KUKA KRL program: MyProgram_116().src

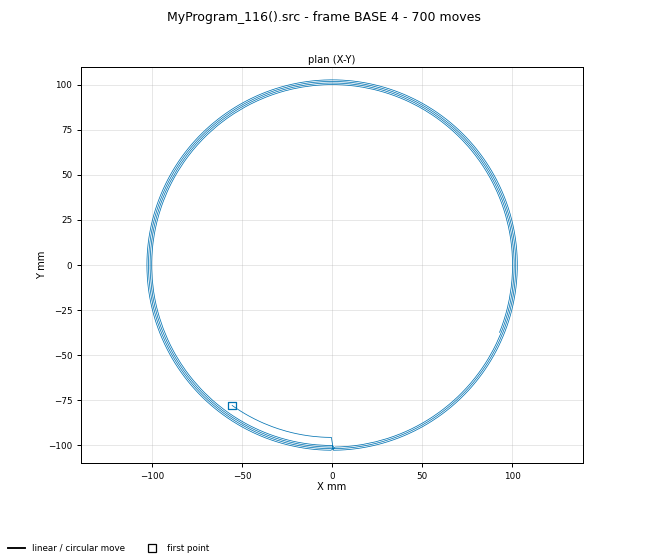
[picture p0: tool path of MyProgram_116().src in frame BASE 4, 700 of 700 moves have a stored position in this frame; points joined in program order, loops and branches not executed]
&ACCESS RVP
&REL 1
&PARAM TEMPLATE = C:\KRC\Roboter\Template\vorgabe
&PARAM EDITMASK = *
DEF MyProgram_116()
; ---- Setting reference (Base) ----
$BASE = BASE_DATA[4]

; --------------------------
; ---- Setting tool (TCP) ----
$TOOL = TOOL_DATA[3]
; --------------------------

$VEL.CP = VEL_APROX_PRINT
Startdeposition()
$VEL.CP = VEL_PRINT
LIN {X -55.4095,Y -77.8597,Z 99,A -129.4251,B 24.9347,C -1.8661,E1 24.9084,E2 214.7041} C_DIS
LIN {X -53.0962,Y -79.4573,Z 99,A -127.8078,B 24.9351,C -1.8611,E1 24.9121,E2 213.0935} C_DIS
LIN {X -50.3768,Y -81.2071,Z 99,A -125.8595,B 24.9353,C -1.8584,E1 24.9167,E2 211.1452} C_DIS
LIN {X -48.3524,Y -82.4286,Z 99,A -124.4407,B 24.9353,C -1.8564,E1 24.9201,E2 209.7269} C_DIS
LIN {X -46.0787,Y -83.7223,Z 99,A -122.868,B 24.9355,C -1.8544,E1 24.9239,E2 208.1545} C_DIS
LIN {X -42.9713,Y -85.3589,Z 99,A -120.7555,B 24.9357,C -1.8519,E1 24.9292,E2 206.042} C_DIS
LIN {X -40.0549,Y -86.7642,Z 99,A -118.7797,B 24.9357,C -1.8509,E1 24.9341,E2 204.0638} C_DIS
LIN {X -37.783,Y -87.778,Z 99,A -117.3046,B 24.9359,C -1.8487,E1 24.9379,E2 202.5903} C_DIS
LIN {X -35.4871,Y -88.7318,Z 99,A -115.8209,B 24.9361,C -1.847,E1 24.9417,E2 201.1074} C_DIS
LIN {X -33.3081,Y -89.5725,Z 99,A -114.4196,B 24.9361,C -1.8457,E1 24.9454,E2 199.7061} C_DIS
LIN {X -29.9786,Y -90.7411,Z 99,A -112.2978,B 24.9363,C -1.8442,E1 24.951,E2 197.5839} C_DIS
LIN {X -27.7453,Y -91.4487,Z 99,A -110.8917,B 24.9363,C -1.8432,E1 24.9548,E2 196.1778} C_DIS
LIN {X -25.4955,Y -92.1013,Z 99,A -109.4857,B 24.9363,C -1.8423,E1 24.9585,E2 194.7716} C_DIS
LIN {X -22.0782,Y -92.9797,Z 99,A -107.3681,B 24.9365,C -1.8412,E1 24.9643,E2 192.6536} C_DIS
LIN {X -19.7944,Y -93.4925,Z 99,A -105.9617,B 24.9365,C -1.8407,E1 24.9681,E2 191.2467} C_DIS
LIN {X -16.3468,Y -94.1565,Z 99,A -103.8547,B 24.9365,C -1.84,E1 24.9739,E2 189.1391} C_DIS
LIN {X -13.1497,Y -94.6546,Z 99,A -101.8803,B 24.9365,C -1.8407,E1 24.9794,E2 187.1612} C_DIS
LIN {X -10.5338,Y -94.9827,Z 99,A -100.3324,B 24.9365,C -1.8393,E1 24.9837,E2 185.6157} C_DIS
LIN {X -8.2054,Y -95.2121,Z 99,A -98.9301,B 24.9365,C -1.8393,E1 24.9876,E2 184.2129} C_DIS
LIN {X -6.146,Y -95.3659,Z 99,A -97.6617,B 24.9365,C -1.8403,E1 24.9911,E2 182.9415} C_DIS
LIN {X -3.7954,Y -95.4883,Z 99,A -96.2517,B 24.9365,C -1.8404,E1 24.995,E2 181.5309} C_DIS
LIN {X -0.3905,Y -95.5626,Z 99,A -94.2196,B 24.9365,C -1.8404,E1 25.0007,E2 179.4987} C_DIS
LIN {X -0.3905,Y -95.5626,Z 99,A -94.2196,B 24.9365,C -1.8404,E1 25.0007,E2 179.4987} C_DIS
Enddeposition()
LIN {X 0.7142,Y -102.6796,Z 100,A -93.2749,B 24.9435,C -1.7358,E1 25.0027,E2 178.8022} C_DIS
Startdeposition()
$VEL.CP = VEL_PRINT
LIN {X 4.3511,Y -102.5901,Z 100,A -91.2947,B 24.9436,C -1.7345,E1 25.0082,E2 176.8254} C_DIS
LIN {X 7.5539,Y -102.406,Z 100,A -89.3348,B 24.9431,C -1.7419,E1 25.0137,E2 174.8488} C_DIS
LIN {X 10.7491,Y -102.1182,Z 100,A -87.6564,B 24.9434,C -1.7386,E1 25.0183,E2 173.1795} C_DIS
LIN {X 13.8193,Y -101.7501,Z 100,A -86.0246,B 24.9435,C -1.7359,E1 25.0228,E2 171.5552} C_DIS
LIN {X 16.3122,Y -101.3803,Z 100,A -84.614,B 24.9435,C -1.7371,E1 25.0267,E2 170.1431} C_DIS
LIN {X 19.3571,Y -100.8413,Z 100,A -82.8685,B 24.9433,C -1.7394,E1 25.0315,E2 168.3943} C_DIS
LIN {X 22.4982,Y -100.1892,Z 100,A -80.9107,B 24.9428,C -1.7476,E1 25.0369,E2 166.4195} C_DIS
LIN {X 25.5043,Y -99.4645,Z 100,A -79.3897,B 24.9432,C -1.7413,E1 25.041,E2 164.9158} C_DIS
LIN {X 28.0492,Y -98.777,Z 100,A -77.8313,B 24.9428,C -1.7463,E1 25.0452,E2 163.348} C_DIS
LIN {X 31.0113,Y -97.8895,Z 100,A -76.2013,B 24.943,C -1.7445,E1 25.0495,E2 161.7252} C_DIS
LIN {X 33.944,Y -96.9096,Z 100,A -74.4511,B 24.9428,C -1.7477,E1 25.0542,E2 159.9708} C_DIS
LIN {X 36.9556,Y -95.8037,Z 100,A -72.5014,B 24.9422,C -1.7565,E1 25.0593,E2 158.0045} C_DIS
LIN {X 39.8227,Y -94.6457,Z 100,A -70.9753,B 24.9425,C -1.751,E1 25.0632,E2 156.495} C_DIS
LIN {X 42.2392,Y -93.5923,Z 100,A -69.4185,B 24.9422,C -1.7567,E1 25.0672,E2 154.9285} C_DIS
LIN {X 45.5515,Y -92.0256,Z 100,A -67.3851,B 24.942,C -1.7596,E1 25.0723,E2 152.8938} C_DIS
LIN {X 48.405,Y -90.5594,Z 100,A -65.6879,B 24.942,C -1.7588,E1 25.0765,E2 151.2031} C_DIS
LIN {X 50.6129,Y -89.3442,Z 100,A -64.2871,B 24.9419,C -1.7611,E1 25.0799,E2 149.801} C_DIS
LIN {X 53.2791,Y -87.7781,Z 100,A -62.5689,B 24.9417,C -1.764,E1 25.084,E2 148.0812} C_DIS
LIN {X 55.5149,Y -86.3815,Z 100,A -61.0131,B 24.9413,C -1.7703,E1 25.0877,E2 146.5155} C_DIS
LIN {X 58.5615,Y -84.3458,Z 100,A -59.0387,B 24.9412,C -1.7715,E1 25.0923,E2 144.5449} C_DIS
LIN {X 61.1689,Y -82.4768,Z 100,A -57.286,B 24.941,C -1.7737,E1 25.0962,E2 142.7933} C_DIS
LIN {X 63.5218,Y -80.6764,Z 100,A -55.5728,B 24.9406,C -1.7798,E1 25.1,E2 141.072} C_DIS
LIN {X 66.1114,Y -78.5706,Z 100,A -53.587,B 24.94,C -1.789,E1 25.1043,E2 139.0721} C_DIS
LIN {X 68.5323,Y -76.4656,Z 100,A -51.9152,B 24.94,C -1.7883,E1 25.1078,E2 137.4086} C_DIS
LIN {X 71.0991,Y -74.0852,Z 100,A -49.9841,B 24.9398,C -1.792,E1 25.1117,E2 135.4766} C_DIS
LIN {X 73.4943,Y -71.7122,Z 100,A -48.191,B 24.9398,C -1.7929,E1 25.1153,E2 133.6889} C_DIS
LIN {X 75.6188,Y -69.4655,Z 100,A -46.4342,B 24.9394,C -1.7986,E1 25.1186,E2 131.9264} C_DIS
LIN {X 77.7534,Y -67.0706,Z 100,A -44.4949,B 24.9386,C -1.8094,E1 25.1222,E2 129.9704} C_DIS
LIN {X 79.7362,Y -64.6978,Z 100,A -42.9791,B 24.9389,C -1.8053,E1 25.1249,E2 128.4713} C_DIS
LIN {X 81.2999,Y -62.7215,Z 100,A -41.5516,B 24.9386,C -1.8099,E1 25.1273,E2 127.0396} C_DIS
LIN {X 83.2212,Y -60.1522,Z 100,A -39.6726,B 24.938,C -1.8185,E1 25.1304,E2 125.1494} C_DIS
LIN {X 84.9931,Y -57.6181,Z 100,A -38.0863,B 24.938,C -1.8175,E1 25.1329,E2 123.5732} C_DIS
LIN {X 86.3815,Y -55.5149,Z 100,A -36.6593,B 24.9377,C -1.8224,E1 25.1351,E2 122.1418} C_DIS
LIN {X 88.0752,Y -52.7903,Z 100,A -34.7097,B 24.9369,C -1.8341,E1 25.138,E2 120.1745} C_DIS
LIN {X 89.6231,Y -50.1134,Z 100,A -33.1655,B 24.9371,C -1.8316,E1 25.1401,E2 118.6442} C_DIS
LIN {X 91.1466,Y -47.2901,Z 100,A -31.4161,B 24.9369,C -1.8352,E1 25.1424,E2 116.8955} C_DIS
LIN {X 92.5275,Y -44.5234,Z 100,A -29.702,B 24.9365,C -1.8399,E1 25.1445,E2 115.1795} C_DIS
LIN {X 93.5923,Y -42.2392,Z 100,A -28.2755,B 24.9362,C -1.845,E1 25.1462,E2 113.7487} C_DIS
LIN {X 94.8679,Y -39.2956,Z 100,A -26.5265,B 24.9359,C -1.8488,E1 25.1481,E2 112.0004} C_DIS
LIN {X 95.8037,Y -36.9556,Z 100,A -24.93,B 24.9351,C -1.8611,E1 25.1497,E2 110.3838} C_DIS
LIN {X 96.9096,Y -33.944,Z 100,A -23.2609,B 24.9351,C -1.8616,E1 25.1513,E2 108.7228} C_DIS
LIN {X 97.8895,Y -31.0113,Z 100,A -21.4381,B 24.9344,C -1.8711,E1 25.1528,E2 106.888} C_DIS
LIN {X 98.777,Y -28.0492,Z 100,A -19.8946,B 24.9345,C -1.8689,E1 25.154,E2 105.3584} C_DIS
LIN {X 99.6069,Y -24.9502,Z 100,A -17.9906,B 24.9338,C -1.8794,E1 25.1554,E2 103.4408} C_DIS
LIN {X 100.3112,Y -21.9393,Z 100,A -16.4325,B 24.9338,C -1.8779,E1 25.1563,E2 101.8951} C_DIS
LIN {X 100.8413,Y -19.3571,Z 100,A -14.8812,B 24.9333,C -1.886,E1 25.1572,E2 100.3339} C_DIS
LIN {X 101.4677,Y -15.7469,Z 100,A -12.8865,B 24.933,C -1.8905,E1 25.1581,E2 98.3403} C_DIS
LIN {X 101.912,Y -12.5696,Z 100,A -10.9641,B 24.9322,C -1.9018,E1 25.1588,E2 96.4025} C_DIS
LIN {X 102.253,Y -9.3797,Z 100,A -9.2954,B 24.9322,C -1.9025,E1 25.1592,E2 94.7421} C_DIS
LIN {X 102.5226,Y -5.7255,Z 100,A -7.3261,B 24.9319,C -1.9059,E1 25.1596,E2 92.7763} C_DIS
LIN {X 102.6533,Y -2.52,Z 100,A -5.5778,B 24.9316,C -1.9099,E1 25.1598,E2 91.029} C_DIS
LIN {X 102.6658,Y 1.8399,Z 100,A -3.1348,B 24.931,C -1.9183,E1 25.1598,E2 88.5808} C_DIS
LIN {X 102.5606,Y 5.0385,Z 100,A -1.2021,B 24.9302,C -1.9301,E1 25.1595,E2 86.6317} C_DIS
LIN {X 102.3604,Y 8.1242,Z 100,A 0.3545,B 24.9302,C -1.9286,E1 25.1592,E2 85.0879} C_DIS
LIN {X 102.0586,Y 11.3181,Z 100,A 2.103,B 24.93,C -1.9325,E1 25.1587,E2 83.3405} C_DIS
LIN {X 101.6696,Y 14.3857,Z 100,A 3.8167,B 24.9296,C -1.9375,E1 25.1581,E2 81.6251} C_DIS
LIN {X 101.286,Y 16.8765,Z 100,A 5.2133,B 24.9293,C -1.9416,E1 25.1574,E2 80.2272} C_DIS
LIN {X 100.8413,Y 19.3571,Z 100,A 6.6896,B 24.9288,C -1.9489,E1 25.1567,E2 78.7422} C_DIS
LIN {X 100.1892,Y 22.4982,Z 100,A 8.5878,B 24.9281,C -1.959,E1 25.1556,E2 76.8314} C_DIS
LIN {X 99.4645,Y 25.5043,Z 100,A 10.1428,B 24.9281,C -1.9572,E1 25.1545,E2 75.2894} C_DIS
LIN {X 98.6211,Y 28.5996,Z 100,A 12.0792,B 24.9273,C -1.9687,E1 25.153,E2 73.337} C_DIS
LIN {X 97.6777,Y 31.6659,Z 100,A 13.7497,B 24.9273,C -1.9691,E1 25.1516,E2 71.6749} C_DIS
LIN {X 96.4857,Y 35.1307,Z 100,A 15.7578,B 24.927,C -1.9737,E1 25.1498,E2 69.6673} C_DIS
LIN {X 95.343,Y 38.1284,Z 100,A 17.6692,B 24.9262,C -1.9839,E1 25.1478,E2 67.7424} C_DIS
LIN {X 94.1036,Y 41.0875,Z 100,A 19.339,B 24.9262,C -1.9842,E1 25.146,E2 66.0812} C_DIS
LIN {X 92.8255,Y 43.9032,Z 100,A 21.1632,B 24.9255,C -1.9931,E1 25.1438,E2 64.2458} C_DIS
LIN {X 91.3057,Y 46.9788,Z 100,A 22.9045,B 24.9257,C -1.9913,E1 25.1416,E2 62.518} C_DIS
LIN {X 89.9586,Y 49.5127,Z 100,A 24.6576,B 24.9249,C -2.0019,E1 25.1393,E2 60.749} C_DIS
LIN {X 88.4253,Y 52.1979,Z 100,A 26.173,B 24.9252,C -1.9979,E1 25.1372,E2 59.2508} C_DIS
LIN {X 87.1177,Y 54.3523,Z 100,A 27.6426,B 24.9247,C -2.0043,E1 25.135,E2 57.7738} C_DIS
LIN {X 85.3788,Y 57.0483,Z 100,A 29.3516,B 24.9246,C -2.0055,E1 25.1324,E2 56.0704} C_DIS
LIN {X 83.9531,Y 59.1264,Z 100,A 30.9333,B 24.9238,C -2.0163,E1 25.1298,E2 54.4711} C_DIS
LIN {X 82.1332,Y 61.6263,Z 100,A 32.4958,B 24.924,C -2.0139,E1 25.1273,E2 52.9216} C_DIS
LIN {X 80.1694,Y 64.1632,Z 100,A 34.2472,B 24.9237,C -2.0166,E1 25.1242,E2 51.1721} C_DIS
LIN {X 78.5706,Y 66.1114,Z 100,A 35.7514,B 24.9232,C -2.0239,E1 25.1215,E2 49.6576} C_DIS
LIN {X 76.5429,Y 68.4459,Z 100,A 37.3928,B 24.9232,C -2.0244,E1 25.1185,E2 48.0222} C_DIS
LIN {X 74.3688,Y 70.805,Z 100,A 39.145,B 24.923,C -2.0268,E1 25.1152,E2 46.272} C_DIS
LIN {X 72.6087,Y 72.6087,Z 100,A 40.7449,B 24.9221,C -2.0377,E1 25.112,E2 44.6532} C_DIS
LIN {X 70.3037,Y 74.8401,Z 100,A 42.4174,B 24.9222,C -2.0367,E1 25.1086,E2 42.99} C_DIS
LIN {X 68.0197,Y 76.9245,Z 100,A 44.0445,B 24.9222,C -2.0362,E1 25.1053,E2 41.3707} C_DIS
LIN {X 66.1114,Y 78.5706,Z 100,A 45.6453,B 24.9214,C -2.0467,E1 25.1018,E2 39.7512} C_DIS
LIN {X 63.6234,Y 80.596,Z 100,A 47.3187,B 24.9216,C -2.0454,E1 25.0982,E2 38.0872} C_DIS
LIN {X 60.7074,Y 82.8147,Z 100,A 49.3424,B 24.9213,C -2.0482,E1 25.0937,E2 36.0642} C_DIS
LIN {X 58.0917,Y 84.6723,Z 100,A 51.0483,B 24.9213,C -2.0478,E1 25.0898,E2 34.3651} C_DIS
LIN {X 55.9963,Y 86.0725,Z 100,A 52.6542,B 24.9206,C -2.058,E1 25.086,E2 32.7403} C_DIS
LIN {X 53.3782,Y 87.7179,Z 100,A 54.1694,B 24.921,C -2.0523,E1 25.0824,E2 31.2434} C_DIS
LIN {X 51.1089,Y 89.0592,Z 100,A 55.7268,B 24.9206,C -2.0578,E1 25.0786,E2 29.6776} C_DIS
LIN {X 47.9683,Y 90.7894,Z 100,A 57.6535,B 24.9206,C -2.0576,E1 25.0739,E2 27.757} C_DIS
LIN {X 45.5515,Y 92.0256,Z 100,A 59.2321,B 24.9203,C -2.0621,E1 25.07,E2 26.1721} C_DIS
LIN {X 42.2392,Y 93.5923,Z 100,A 61.1804,B 24.9203,C -2.0607,E1 25.0651,E2 24.2321} C_DIS
LIN {X 39.9296,Y 94.6007,Z 100,A 62.5833,B 24.9203,C -2.0621,E1 25.0615,E2 22.8292} C_DIS
LIN {X 37.488,Y 95.5945,Z 100,A 64.1425,B 24.9199,C -2.067,E1 25.0574,E2 21.2618} C_DIS
LIN {X 34.5933,Y 96.6817,Z 100,A 65.7733,B 24.92,C -2.0649,E1 25.0531,E2 19.6394} C_DIS
LIN {X 31.6659,Y 97.6777,Z 100,A 67.4956,B 24.92,C -2.0662,E1 25.0486,E2 17.9173} C_DIS
LIN {X 29.232,Y 98.4335,Z 100,A 68.9367,B 24.9198,C -2.068,E1 25.0447,E2 16.4744} C_DIS
LIN {X 26.1707,Y 99.2933,Z 100,A 70.8881,B 24.9192,C -2.076,E1 25.0394,E2 14.5072} C_DIS
LIN {X 23.0556,Y 100.0605,Z 100,A 72.5665,B 24.9194,C -2.0727,E1 25.0349,E2 12.839} C_DIS
LIN {X 20.0327,Y 100.7112,Z 100,A 74.1987,B 24.9197,C -2.0699,E1 25.0304,E2 11.2155} C_DIS
LIN {X 17.5551,Y 101.1725,Z 100,A 75.604,B 24.9197,C -2.0704,E1 25.0266,E2 9.8107} C_DIS
LIN {X 14.5005,Y 101.6533,Z 100,A 77.3579,B 24.9195,C -2.072,E1 25.0217,E2 8.0545} C_DIS
LIN {X 11.3181,Y 102.0586,Z 100,A 79.1177,B 24.9195,C -2.0712,E1 25.0169,E2 6.2981} C_DIS
LIN {X 8.81,Y 102.3056,Z 100,A 80.5236,B 24.9195,C -2.0712,E1 25.013,E2 4.8927} C_DIS
LIN {X 5.7255,Y 102.5226,Z 100,A 82.2787,B 24.9195,C -2.0725,E1 25.0081,E2 3.1355} C_DIS
LIN {X 2.52,Y 102.6533,Z 100,A 84.2409,B 24.919,C -2.0788,E1 25.0025,E2 1.1587} C_DIS
LIN {X -0.733,Y 102.6797,Z 100,A 85.9351,B 24.9193,C -2.0739,E1 24.9978,E2 -0.5237} C_DIS
LIN {X -4.3511,Y 102.5901,Z 100,A 87.906,B 24.9195,C -2.0715,E1 24.9924,E2 -2.4892} C_DIS
LIN {X -7.5539,Y 102.406,Z 100,A 89.8698,B 24.9191,C -2.0772,E1 24.9868,E2 -4.4674} C_DIS
LIN {X -10.7491,Y 102.1182,Z 100,A 91.5519,B 24.9195,C -2.0723,E1 24.9822,E2 -6.1386} C_DIS
LIN {X -13.8193,Y 101.7501,Z 100,A 93.1879,B 24.9198,C -2.0679,E1 24.9777,E2 -7.7654} C_DIS
LIN {X -16.3122,Y 101.3803,Z 100,A 94.5963,B 24.9198,C -2.067,E1 24.9738,E2 -9.1729} C_DIS
LIN {X -19.3571,Y 100.8413,Z 100,A 96.4073,B 24.9198,C -2.0689,E1 24.9688,E2 -10.9903} C_DIS
LIN {X -22.4982,Y 100.1892,Z 100,A 98.3201,B 24.9195,C -2.0718,E1 24.9636,E2 -12.9125} C_DIS
LIN {X -25.5043,Y 99.4645,Z 100,A 99.8474,B 24.9202,C -2.0629,E1 24.9595,E2 -14.4206} C_DIS
LIN {X -28.1373,Y 98.7521,Z 100,A 101.4409,B 24.9202,C -2.0639,E1 24.9552,E2 -16.019} C_DIS
LIN {X -31.5555,Y 97.7134,Z 100,A 103.3711,B 24.9205,C -2.0593,E1 24.9501,E2 -17.9417} C_DIS
LIN {X -33.944,Y 96.9096,Z 100,A 104.811,B 24.9205,C -2.0588,E1 24.9463,E2 -19.3831} C_DIS
LIN {X -36.9556,Y 95.8037,Z 100,A 106.5767,B 24.9208,C -2.0555,E1 24.9417,E2 -21.1447} C_DIS
LIN {X -39.8227,Y 94.6457,Z 100,A 108.3075,B 24.9209,C -2.0533,E1 24.9372,E2 -22.8742} C_DIS
LIN {X -42.2392,Y 93.5923,Z 100,A 109.8748,B 24.9209,C -2.0546,E1 24.9332,E2 -24.4484} C_DIS
LIN {X -45.5515,Y 92.0256,Z 100,A 111.8645,B 24.9212,C -2.0494,E1 24.9282,E2 -26.4308} C_DIS
LIN {X -48.405,Y 90.5594,Z 100,A 113.6318,B 24.9215,C -2.0456,E1 24.9238,E2 -28.1938} C_DIS
LIN {X -51.1089,Y 89.0592,Z 100,A 115.3635,B 24.9217,C -2.0428,E1 24.9196,E2 -29.924} C_DIS
LIN {X -53.3782,Y 87.7179,Z 100,A 116.9323,B 24.9217,C -2.0437,E1 24.9158,E2 -31.4996} C_DIS
LIN {X -55.9963,Y 86.0725,Z 100,A 118.7753,B 24.9217,C -2.0446,E1 24.9115,E2 -33.3508} C_DIS
LIN {X -58.5615,Y 84.3458,Z 100,A 120.3059,B 24.9224,C -2.0342,E1 24.908,E2 -34.8618} C_DIS
LIN {X -60.6138,Y 82.8832,Z 100,A 121.7185,B 24.9226,C -2.0316,E1 24.9048,E2 -36.273} C_DIS
LIN {X -62.7215,Y 81.2999,Z 100,A 123.2882,B 24.9226,C -2.032,E1 24.9013,E2 -37.8494} C_DIS
LIN {X -65.5822,Y 79.0104,Z 100,A 125.2504,B 24.9231,C -2.0246,E1 24.8971,E2 -39.8014} C_DIS
LIN {X -67.5014,Y 77.3771,Z 100,A 126.6936,B 24.9233,C -2.0227,E1 24.894,E2 -41.2459} C_DIS
LIN {X -69.887,Y 75.2321,Z 100,A 128.6461,B 24.9232,C -2.0243,E1 24.89,E2 -43.2101} C_DIS
LIN {X -72.1192,Y 73.0923,Z 100,A 130.1975,B 24.9239,C -2.0141,E1 24.8869,E2 -44.7434} C_DIS
LIN {X -73.9718,Y 71.2168,Z 100,A 131.7681,B 24.9239,C -2.0141,E1 24.8838,E2 -46.3206} C_DIS
LIN {X -76.084,Y 68.9585,Z 100,A 133.4111,B 24.9245,C -2.0067,E1 24.8808,E2 -47.9536} C_DIS
LIN {X -77.7534,Y 67.0706,Z 100,A 135.0318,B 24.9242,C -2.0107,E1 24.8778,E2 -49.5911} C_DIS
LIN {X -79.7362,Y 64.6978,Z 100,A 136.5904,B 24.925,C -2.0004,E1 24.875,E2 -51.1322} C_DIS
LIN {X -81.7199,Y 62.1764,Z 100,A 138.5638,B 24.9248,C -2.002,E1 24.8716,E2 -53.119} C_DIS
LIN {X -83.5535,Y 59.6865,Z 100,A 140.097,B 24.9257,C -1.9906,E1 24.8692,E2 -54.6322} C_DIS
LIN {X -85.0581,Y 57.522,Z 100,A 141.6688,B 24.9257,C -1.9901,E1 24.8667,E2 -56.2106} C_DIS
LIN {X -86.7532,Y 54.9358,Z 100,A 143.3129,B 24.9263,C -1.9823,E1 24.8642,E2 -57.8446} C_DIS
LIN {X -88.3663,Y 52.2978,Z 100,A 145.0791,B 24.9266,C -1.9788,E1 24.8616,E2 -59.6115} C_DIS
LIN {X -89.9586,Y 49.5127,Z 100,A 146.8506,B 24.927,C -1.9729,E1 24.8592,E2 -61.3783} C_DIS
LIN {X -91.1466,Y 47.2901,Z 100,A 148.2661,B 24.9273,C -1.9691,E1 24.8574,E2 -62.7922} C_DIS
LIN {X -92.2797,Y 45.039,Z 100,A 149.8841,B 24.9271,C -1.9724,E1 24.8554,E2 -64.4267} C_DIS
LIN {X -93.7408,Y 41.9096,Z 100,A 151.656,B 24.9279,C -1.9612,E1 24.8533,E2 -66.1815} C_DIS
LIN {X -95.0835,Y 38.7657,Z 100,A 153.5418,B 24.9284,C -1.9546,E1 24.8513,E2 -68.0621} C_DIS
LIN {X -96.0063,Y 36.4206,Z 100,A 154.9716,B 24.9286,C -1.9511,E1 24.8499,E2 -69.4916} C_DIS
LIN {X -96.9096,Y 33.944,Z 100,A 156.5304,B 24.9287,C -1.9496,E1 24.8484,E2 -71.0557} C_DIS
LIN {X -97.8895,Y 31.0113,Z 100,A 158.3783,B 24.9288,C -1.9484,E1 24.8468,E2 -72.9115} C_DIS
LIN {X -98.777,Y 28.0492,Z 100,A 159.9515,B 24.9296,C -1.9377,E1 24.8456,E2 -74.4682} C_DIS
LIN {X -99.6069,Y 24.9502,Z 100,A 161.9185,B 24.9296,C -1.9382,E1 24.8442,E2 -76.4478} C_DIS
LIN {X -100.3359,Y 21.826,Z 100,A 163.6104,B 24.9302,C -1.9291,E1 24.8432,E2 -78.1279} C_DIS
LIN {X -101.0507,Y 18.2323,Z 100,A 165.6071,B 24.9308,C -1.9209,E1 24.8421,E2 -80.1168} C_DIS
LIN {X -101.5728,Y 15.0669,Z 100,A 167.5828,B 24.9308,C -1.9216,E1 24.8413,E2 -82.106} C_DIS
LIN {X -101.9786,Y 12.0015,Z 100,A 169.1175,B 24.9317,C -1.9094,E1 24.8408,E2 -83.6208} C_DIS
LIN {X -102.2424,Y 9.4952,Z 100,A 170.5637,B 24.9319,C -1.9063,E1 24.8404,E2 -85.0681} C_DIS
LIN {X -102.491,Y 6.2967,Z 100,A 172.3365,B 24.9323,C -1.8999,E1 24.84,E2 -86.8364} C_DIS
LIN {X -102.6322,Y 3.2077,Z 100,A 174.1042,B 24.9326,C -1.8958,E1 24.8398,E2 -88.605} C_DIS
LIN {X -102.6841,Y 0,Z 100,A 176.0769,B 24.9326,C -1.8964,E1 24.8398,E2 -90.5909} C_DIS
LIN {X -102.6322,Y -3.2077,Z 100,A 177.7719,B 24.9332,C -1.8873,E1 24.8399,E2 -92.2746} C_DIS
LIN {X -102.4524,Y -6.8674,Z 100,A 179.739,B 24.9339,C -1.8781,E1 24.8402,E2 -94.2315} C_DIS
LIN {X -102.253,Y -9.3797,Z 100,A -178.8154,B 24.9341,C -1.875,E1 24.8406,E2 -95.6783} C_DIS
LIN {X -101.912,Y -12.5696,Z 100,A -177.0425,B 24.9345,C -1.8686,E1 24.8411,E2 -97.4467} C_DIS
LIN {X -101.5728,Y -15.0669,Z 100,A -175.6264,B 24.9348,C -1.8646,E1 24.8417,E2 -98.8615} C_DIS
LIN {X -101.1725,Y -17.5551,Z 100,A -174.0078,B 24.9346,C -1.8676,E1 24.8424,E2 -100.497} C_DIS
LIN {X -100.5728,Y -20.7067,Z 100,A -172.3163,B 24.9352,C -1.8586,E1 24.8434,E2 -102.177} C_DIS
LIN {X -99.77,Y -24.2818,Z 100,A -170.3499,B 24.9359,C -1.8495,E1 24.8446,E2 -104.1333} C_DIS
LIN {X -99.1441,Y -26.723,Z 100,A -168.9042,B 24.9361,C -1.8466,E1 24.8456,E2 -105.5805} C_DIS
LIN {X -98.2627,Y -29.8077,Z 100,A -167.1318,B 24.9365,C -1.8405,E1 24.847,E2 -107.3486} C_DIS
LIN {X -97.4709,Y -32.3013,Z 100,A -165.498,B 24.9364,C -1.8423,E1 24.8484,E2 -108.9959} C_DIS
LIN {X -96.446,Y -35.2397,Z 100,A -163.8227,B 24.9369,C -1.835,E1 24.85,E2 -110.6634} C_DIS
LIN {X -95.3429,Y -38.1284,Z 100,A -161.9757,B 24.9369,C -1.8342,E1 24.8519,E2 -112.5189} C_DIS
LIN {X -94.1499,Y -40.9812,Z 100,A -160.412,B 24.9377,C -1.8236,E1 24.8536,E2 -114.0658} C_DIS
LIN {X -92.8255,Y -43.9032,Z 100,A -158.438,B 24.9376,C -1.825,E1 24.856,E2 -116.0541} C_DIS
LIN {X -91.4069,Y -46.7807,Z 100,A -156.7477,B 24.9381,C -1.8165,E1 24.8581,E2 -117.7332} C_DIS
LIN {X -89.9586,Y -49.5127,Z 100,A -155.104,B 24.9387,C -1.8089,E1 24.8602,E2 -119.3674} C_DIS
LIN {X -88.7057,Y -51.7235,Z 100,A -153.4836,B 24.9384,C -1.8123,E1 24.8625,E2 -121.0044} C_DIS
LIN {X -87.1177,Y -54.3523,Z 100,A -151.9241,B 24.9391,C -1.8023,E1 24.8648,E2 -122.5481} C_DIS
LIN {X -85.3788,Y -57.0483,Z 100,A -149.9513,B 24.939,C -1.8042,E1 24.8678,E2 -124.5353} C_DIS
LIN {X -83.5535,Y -59.6865,Z 100,A -148.2619,B 24.9395,C -1.7962,E1 24.8705,E2 -126.2138} C_DIS
LIN {X -81.7199,Y -62.1764,Z 100,A -146.619,B 24.94,C -1.789,E1 24.8733,E2 -127.8473} C_DIS
LIN {X -80.1694,Y -64.1632,Z 100,A -145.2057,B 24.9402,C -1.7858,E1 24.8757,E2 -129.2599} C_DIS
LIN {X -78.1996,Y -66.5468,Z 100,A -143.4711,B 24.9405,C -1.7822,E1 24.8788,E2 -130.9938} C_DIS
LIN {X -76.4656,Y -68.5323,Z 100,A -141.9013,B 24.9405,C -1.7824,E1 24.8817,E2 -132.5712} C_DIS
LIN {X -74.081,Y -71.1035,Z 100,A -139.9496,B 24.9408,C -1.778,E1 24.8855,E2 -134.5208} C_DIS
LIN {X -71.7122,Y -73.4943,Z 100,A -138.1401,B 24.9412,C -1.7715,E1 24.889,E2 -136.3225} C_DIS
LIN {X -69.4655,Y -75.6188,Z 100,A -136.3373,B 24.9412,C -1.7708,E1 24.8927,E2 -138.131} C_DIS
LIN {X -67.0706,Y -77.7534,Z 100,A -134.4072,B 24.9412,C -1.7724,E1 24.8968,E2 -140.0725} C_DIS
LIN {X -64.6978,Y -79.7362,Z 100,A -132.8767,B 24.9418,C -1.7621,E1 24.9001,E2 -141.5843} C_DIS
LIN {X -62.7215,Y -81.2999,Z 100,A -131.3942,B 24.9418,C -1.7623,E1 24.9034,E2 -143.0728} C_DIS
LIN {X -60.1522,Y -83.2212,Z 100,A -129.6678,B 24.9422,C -1.7569,E1 24.9072,E2 -144.7923} C_DIS
LIN {X -57.6181,Y -84.9931,Z 100,A -127.9364,B 24.9423,C -1.7543,E1 24.9112,E2 -146.5235} C_DIS
LIN {X -55.3837,Y -86.4657,Z 100,A -126.357,B 24.9423,C -1.7551,E1 24.9149,E2 -148.11} C_DIS
LIN {X -52.2978,Y -88.3663,Z 100,A -124.4092,B 24.9426,C -1.7494,E1 24.9195,E2 -150.0501} C_DIS
LIN {X -50.1134,Y -89.6231,Z 100,A -122.9688,B 24.9426,C -1.7487,E1 24.9231,E2 -151.4931} C_DIS
LIN {X -47.2901,Y -91.1466,Z 100,A -121.2031,B 24.9429,C -1.7454,E1 24.9274,E2 -153.2559} C_DIS
LIN {X -44.5234,Y -92.5275,Z 100,A -119.4734,B 24.943,C -1.7435,E1 24.9317,E2 -154.9856} C_DIS
LIN {X -42.2392,Y -93.5923,Z 100,A -118.0339,B 24.943,C -1.7432,E1 24.9354,E2 -156.4278} C_DIS
LIN {X -39.2956,Y -94.8679,Z 100,A -116.2179,B 24.9431,C -1.7422,E1 24.9401,E2 -158.2458} C_DIS
LIN {X -36.9556,Y -95.8037,Z 100,A -114.6586,B 24.9428,C -1.7466,E1 24.9442,E2 -159.8189} C_DIS
LIN {X -33.944,Y -96.9096,Z 100,A -112.9751,B 24.9432,C -1.7411,E1 24.9486,E2 -161.4925} C_DIS
LIN {X -31.0113,Y -97.8895,Z 100,A -111.1367,B 24.943,C -1.744,E1 24.9535,E2 -163.3412} C_DIS
LIN {X -28.0492,Y -98.777,Z 100,A -109.5804,B 24.9435,C -1.7364,E1 24.9576,E2 -164.8821} C_DIS
LIN {X -24.9502,Y -99.6069,Z 100,A -107.6799,B 24.9433,C -1.7396,E1 24.9628,E2 -166.7928} C_DIS
LIN {X -21.9393,Y -100.3112,Z 100,A -106.0296,B 24.9435,C -1.7359,E1 24.9673,E2 -168.4365} C_DIS
LIN {X -18.7953,Y -100.9494,Z 100,A -104.0974,B 24.9432,C -1.7406,E1 24.9726,E2 -170.3821} C_DIS
LIN {X -15.7469,Y -101.4677,Z 100,A -102.5722,B 24.9437,C -1.7325,E1 24.9767,E2 -171.8894} C_DIS
LIN {X -13.137,Y -101.8385,Z 100,A -101.0091,B 24.9435,C -1.7357,E1 24.9811,E2 -173.4613} C_DIS
LIN {X -10.0648,Y -102.1898,Z 100,A -99.3746,B 24.9438,C -1.732,E1 24.9856,E2 -175.088} C_DIS
LIN {X -7.5539,Y -102.406,Z 100,A -97.7672,B 24.9433,C -1.7397,E1 24.9901,E2 -176.7144} C_DIS
LIN {X -4.3511,Y -102.5901,Z 100,A -96.0871,B 24.9435,C -1.7356,E1 24.9948,E2 -178.3852} C_DIS
LIN {X -0.688,Y -102.68,Z 100,A -94.1049,B 24.9437,C -1.7336,E1 25.0003,E2 -180.3627} C_DIS
LIN {X -0.688,Y -102.68,Z 100,A -94.1049,B 24.9437,C -1.7336,E1 25.0003,E2 -180.3627} C_DIS
Enddeposition()
LIN {X 0.7106,Y -101.8004,Z 100,A -93.8606,B 24.944,C -1.7284,E1 25.001,E2 -180.5947} C_DIS
Startdeposition()
$VEL.CP = VEL_PRINT
LIN {X -1.7832,Y -101.7888,Z 100,A -95.4939,B 24.9446,C -1.7194,E1 24.9963,E2 -178.9399} C_DIS
LIN {X -4.8954,Y -101.688,Z 100,A -97.4182,B 24.945,C -1.7127,E1 24.9909,E2 -176.9993} C_DIS
LIN {X -8.8916,Y -101.4164,Z 100,A -99.5623,B 24.9448,C -1.7169,E1 24.985,E2 -174.8643} C_DIS
LIN {X -11.9838,Y -101.0967,Z 100,A -101.2448,B 24.9446,C -1.7196,E1 24.9803,E2 -173.1872} C_DIS
LIN {X -15.0977,Y -100.6797,Z 100,A -103.0687,B 24.9446,C -1.7179,E1 24.9753,E2 -171.3578} C_DIS
LIN {X -18.4337,Y -100.1225,Z 100,A -105.2173,B 24.9452,C -1.7094,E1 24.9693,E2 -169.1869} C_DIS
LIN {X -22.8304,Y -99.2115,Z 100,A -107.4911,B 24.9446,C -1.72,E1 24.9632,E2 -166.9355} C_DIS
LIN {X -26.3709,Y -98.3298,Z 100,A -109.5381,B 24.9445,C -1.7214,E1 24.9576,E2 -164.8888} C_DIS
LIN {X -30.9896,Y -96.9738,Z 100,A -112.0293,B 24.9438,C -1.7314,E1 24.951,E2 -162.4171} C_DIS
LIN {X -33.5048,Y -96.1333,Z 100,A -113.5711,B 24.9438,C -1.7308,E1 24.9469,E2 -160.871} C_DIS
LIN {X -35.9884,Y -95.2312,Z 100,A -115.2838,B 24.9443,C -1.7238,E1 24.9424,E2 -159.1382} C_DIS
LIN {X -39.278,Y -93.9226,Z 100,A -117.2436,B 24.9441,C -1.727,E1 24.9373,E2 -157.1817} C_DIS
LIN {X -42.1981,Y -92.6478,Z 100,A -119.1551,B 24.9443,C -1.7247,E1 24.9324,E2 -155.26} C_DIS
LIN {X -45.4281,Y -91.107,Z 100,A -121.2594,B 24.9443,C -1.7239,E1 24.9271,E2 -153.1482} C_DIS
LIN {X -50.8147,Y -88.2157,Z 100,A -125.1023,B 24.9449,C -1.7142,E1 24.9177,E2 -149.2711} C_DIS
LIN {X -54.1802,Y -86.19,Z 100,A -126.761,B 24.9434,C -1.7372,E1 24.9139,E2 -147.6622} C_DIS
LIN {X -57.0004,Y -84.351,Z 100,A -128.6308,B 24.9432,C -1.7412,E1 24.9095,E2 -145.7955} C_DIS
LIN {X -59.9272,Y -82.2978,Z 100,A -130.7217,B 24.9432,C -1.7417,E1 24.9047,E2 -143.6987} C_DIS
LIN {X -63.1824,Y -79.8256,Z 100,A -133.055,B 24.943,C -1.7447,E1 24.8996,E2 -141.364} C_DIS
LIN {X -65.9201,Y -77.5802,Z 100,A -135.0175,B 24.9426,C -1.7496,E1 24.8954,E2 -139.4055} C_DIS
LIN {X -68.6114,Y -75.211,Z 100,A -136.9618,B 24.9422,C -1.7562,E1 24.8914,E2 -137.4691} C_DIS
LIN {X -71.0775,Y -72.8867,Z 100,A -138.8021,B 24.9418,C -1.7624,E1 24.8877,E2 -135.6362} C_DIS
LIN {X -73.2935,Y -70.6555,Z 100,A -140.6654,B 24.9418,C -1.763,E1 24.884,E2 -133.7661} C_DIS
LIN {X -75.5066,Y -68.2872,Z 100,A -142.6421,B 24.9418,C -1.7616,E1 24.8803,E2 -131.7776} C_DIS
LIN {X -77.4932,Y -66.0222,Z 100,A -144.2698,B 24.9414,C -1.7679,E1 24.8773,E2 -130.1574} C_DIS
LIN {X -79.9863,Y -62.9791,Z 100,A -146.3878,B 24.9408,C -1.7765,E1 24.8736,E2 -128.05} C_DIS
LIN {X -82.0701,Y -60.2383,Z 100,A -148.386,B 24.9407,C -1.7791,E1 24.8703,E2 -126.0485} C_DIS
LIN {X -83.9401,Y -57.607,Z 100,A -150.3236,B 24.9407,C -1.7795,E1 24.8671,E2 -124.1021} C_DIS
LIN {X -85.811,Y -54.7783,Z 100,A -152.2272,B 24.9403,C -1.7846,E1 24.8643,E2 -122.2011} C_DIS
LIN {X -88.0597,Y -51.0862,Z 100,A -154.6013,B 24.9397,C -1.7931,E1 24.8609,E2 -119.8351} C_DIS
LIN {X -89.6413,Y -48.2563,Z 100,A -156.3622,B 24.9393,C -1.8002,E1 24.8585,E2 -118.0819} C_DIS
LIN {X -91.0486,Y -45.5458,Z 100,A -158.1792,B 24.9392,C -1.8016,E1 24.8562,E2 -116.2585} C_DIS
LIN {X -92.5718,Y -42.3669,Z 100,A -160.3616,B 24.9392,C -1.8004,E1 24.8536,E2 -114.0612} C_DIS
LIN {X -94.2617,Y -38.4561,Z 100,A -162.5602,B 24.9383,C -1.8141,E1 24.8512,E2 -111.8832} C_DIS
LIN {X -95.4841,Y -35.3146,Z 100,A -164.5884,B 24.9383,C -1.8152,E1 24.8492,E2 -109.8461} C_DIS
LIN {X -96.74,Y -31.712,Z 100,A -166.8918,B 24.9382,C -1.8163,E1 24.8472,E2 -107.5322} C_DIS
LIN {X -97.9989,Y -27.5751,Z 100,A -169.1255,B 24.9372,C -1.8305,E1 24.8454,E2 -105.3194} C_DIS
LIN {X -98.9062,Y -24.1185,Z 100,A -171.0199,B 24.9365,C -1.8406,E1 24.8441,E2 -103.4382} C_DIS
LIN {X -99.6248,Y -20.9589,Z 100,A -173.0019,B 24.9365,C -1.8409,E1 24.8429,E2 -101.4451} C_DIS
LIN {X -100.2676,Y -17.627,Z 100,A -174.9293,B 24.9361,C -1.8463,E1 24.842,E2 -99.5191} C_DIS
LIN {X -100.9082,Y -13.4849,Z 100,A -177.2216,B 24.9354,C -1.856,E1 24.8411,E2 -97.2363} C_DIS
LIN {X -101.4898,Y -7.9974,Z 100,A 179.5834,B 24.935,C -1.8628,E1 24.8402,E2 -94.0385} C_DIS
LIN {X -101.711,Y -4.3604,Z 100,A 177.5533,B 24.9344,C -1.8701,E1 24.8399,E2 -92.0135} C_DIS
LIN {X -101.8052,Y -0.1706,Z 100,A 174.792,B 24.9349,C -1.864,E1 24.8399,E2 -89.2211} C_DIS
LIN {X -101.7142,Y 4.2858,Z 100,A 172.6458,B 24.9334,C -1.8844,E1 24.8399,E2 -87.1106} C_DIS
LIN {X -101.4501,Y 8.4949,Z 100,A 169.5974,B 24.9345,C -1.8693,E1 24.8407,E2 -84.0079} C_DIS
LIN {X -101.0101,Y 12.6985,Z 100,A 168.1018,B 24.9318,C -1.9067,E1 24.8411,E2 -82.5926} C_DIS
LIN {X -100.4609,Y 16.4876,Z 100,A 165.683,B 24.932,C -1.9047,E1 24.8421,E2 -80.1545} C_DIS
LIN {X -99.8842,Y 19.6844,Z 100,A 163.8522,B 24.9316,C -1.9105,E1 24.8431,E2 -78.3267} C_DIS
LIN {X -99.1886,Y 22.9295,Z 100,A 161.9906,B 24.9311,C -1.9166,E1 24.8442,E2 -76.4688} C_DIS
LIN {X -98.3001,Y 26.4806,Z 100,A 159.9298,B 24.9307,C -1.9231,E1 24.8456,E2 -74.4116} C_DIS
LIN {X -97.3152,Y 29.899,Z 100,A 157.9331,B 24.9302,C -1.9296,E1 24.8472,E2 -72.4188} C_DIS
LIN {X -96.2676,Y 33.121,Z 100,A 155.8458,B 24.9302,C -1.9294,E1 24.8491,E2 -70.3191} C_DIS
LIN {X -94.9166,Y 36.8126,Z 100,A 153.6681,B 24.9296,C -1.9374,E1 24.8512,E2 -68.1482} C_DIS
LIN {X -93.6471,Y 39.9316,Z 100,A 151.8723,B 24.929,C -1.9466,E1 24.8531,E2 -66.3643} C_DIS
LIN {X -92.0391,Y 43.5122,Z 100,A 149.5059,B 24.9289,C -1.9479,E1 24.8559,E2 -63.988} C_DIS
LIN {X -90.4442,Y 46.7353,Z 100,A 147.2105,B 24.9291,C -1.9446,E1 24.8588,E2 -61.6726} C_DIS
LIN {X -87.8969,Y 51.3666,Z 100,A 144.5183,B 24.9278,C -1.9629,E1 24.8625,E2 -59.0098} C_DIS
LIN {X -86.0542,Y 54.3976,Z 100,A 142.462,B 24.9275,C -1.9665,E1 24.8655,E2 -56.9516} C_DIS
LIN {X -84.0925,Y 57.3822,Z 100,A 140.3063,B 24.9275,C -1.9671,E1 24.8689,E2 -54.7867} C_DIS
LIN {X -81.8011,Y 60.6055,Z 100,A 138.4273,B 24.9261,C -1.985,E1 24.8719,E2 -52.9413} C_DIS
LIN {X -80.3277,Y 62.5448,Z 100,A 136.8091,B 24.9265,C -1.9802,E1 24.8747,E2 -51.3039} C_DIS
LIN {X -78.1651,Y 65.2257,Z 100,A 134.8839,B 24.9261,C -1.9857,E1 24.8781,E2 -49.383} C_DIS
LIN {X -75.7031,Y 68.0678,Z 100,A 133.0083,B 24.925,C -1.9994,E1 24.8815,E2 -47.5316} C_DIS
LIN {X -73.9965,Y 69.9193,Z 100,A 131.4877,B 24.925,C -1.9994,E1 24.8844,E2 -46.0042} C_DIS
LIN {X -71.7541,Y 72.2189,Z 100,A 129.6308,B 24.9248,C -2.0021,E1 24.8881,E2 -44.1458} C_DIS
LIN {X -69.5639,Y 74.3308,Z 100,A 127.9314,B 24.9245,C -2.0066,E1 24.8915,E2 -42.45} C_DIS
LIN {X -66.8851,Y 76.7498,Z 100,A 125.8957,B 24.9242,C -2.0111,E1 24.8958,E2 -40.417} C_DIS
LIN {X -64.1878,Y 79.0194,Z 100,A 123.8789,B 24.9239,C -2.0143,E1 24.9001,E2 -38.4002} C_DIS
LIN {X -61.3338,Y 81.2549,Z 100,A 121.8094,B 24.9237,C -2.0176,E1 24.9047,E2 -36.331} C_DIS
LIN {X -58.4452,Y 83.3574,Z 100,A 119.7981,B 24.9234,C -2.0217,E1 24.9092,E2 -34.3224} C_DIS
LIN {X -55.8048,Y 85.1472,Z 100,A 117.9738,B 24.9232,C -2.0241,E1 24.9135,E2 -32.498} C_DIS
LIN {X -52.7494,Y 87.0727,Z 100,A 115.9576,B 24.9228,C -2.0285,E1 24.9183,E2 -30.4859} C_DIS
LIN {X -49.6051,Y 88.9014,Z 100,A 113.9333,B 24.9225,C -2.0329,E1 24.9232,E2 -28.4661} C_DIS
LIN {X -46.2504,Y 90.692,Z 100,A 111.6514,B 24.9226,C -2.0315,E1 24.9288,E2 -26.1745} C_DIS
LIN {X -41.4925,Y 92.9658,Z 100,A 108.9712,B 24.9215,C -2.0463,E1 24.9355,E2 -23.5228} C_DIS
LIN {X -37.1993,Y 94.7647,Z 100,A 106.2948,B 24.9214,C -2.0479,E1 24.9425,E2 -20.8442} C_DIS
LIN {X -34.7896,Y 95.6757,Z 100,A 104.7168,B 24.9216,C -2.0452,E1 24.9466,E2 -19.2566} C_DIS
LIN {X -31.782,Y 96.7174,Z 100,A 102.8411,B 24.9216,C -2.0444,E1 24.9516,E2 -17.3752} C_DIS
LIN {X -28.6309,Y 97.6961,Z 100,A 101.1064,B 24.9211,C -2.0509,E1 24.9562,E2 -15.653} C_DIS
LIN {X -23.0885,Y 99.1518,Z 100,A 97.7523,B 24.9212,C -2.0494,E1 24.9653,E2 -12.2905} C_DIS
LIN {X -20.3319,Y 99.7535,Z 100,A 95.3631,B 24.9233,C -2.0219,E1 24.972,E2 -9.8333} C_DIS
LIN {X -15.5497,Y 100.6099,Z 100,A 93.8875,B 24.9197,C -2.0694,E1 24.9758,E2 -8.4692} C_DIS
LIN {X -13.2343,Y 100.9406,Z 100,A 92.1386,B 24.9209,C -2.0544,E1 24.9807,E2 -6.6832} C_DIS
LIN {X -10.1343,Y 101.2998,Z 100,A 89.9707,B 24.9219,C -2.0403,E1 24.9868,E2 -4.4806} C_DIS
LIN {X -5.3807,Y 101.6624,Z 100,A 87.8413,B 24.9203,C -2.0617,E1 24.9926,E2 -2.4012} C_DIS
LIN {X -2.4627,Y 101.7763,Z 100,A 85.9362,B 24.921,C -2.0525,E1 24.998,E2 -0.474} C_DIS
LIN {X 0.868,Y 101.801,Z 100,A 84.2505,B 24.9204,C -2.0599,E1 25.0026,E2 1.1941} C_DIS
LIN {X 4.1471,Y 101.7201,Z 100,A 82.3166,B 24.9207,C -2.0568,E1 25.0081,E2 3.1349} C_DIS
LIN {X 7.7341,Y 101.5109,Z 100,A 80.3109,B 24.9207,C -2.0573,E1 25.0136,E2 5.1384} C_DIS
LIN {X 11.2839,Y 101.1785,Z 100,A 78.2472,B 24.9208,C -2.0549,E1 25.0194,E2 7.2065} C_DIS
LIN {X 14.335,Y 100.7901,Z 100,A 76.5618,B 24.9208,C -2.0563,E1 25.024,E2 8.8873} C_DIS
LIN {X 18.2861,Y 100.149,Z 100,A 74.2671,B 24.9208,C -2.0539,E1 25.0304,E2 11.1852} C_DIS
LIN {X 21.8166,Y 99.4394,Z 100,A 72.276,B 24.9208,C -2.0543,E1 25.0358,E2 13.1729} C_DIS
LIN {X 27.5615,Y 98.0028,Z 100,A 69.0236,B 24.9208,C -2.0553,E1 25.0446,E2 16.4179} C_DIS
LIN {X 30.5094,Y 97.126,Z 100,A 67.362,B 24.9207,C -2.0566,E1 25.049,E2 18.0734} C_DIS
LIN {X 32.9609,Y 96.322,Z 100,A 65.6695,B 24.9215,C -2.0462,E1 25.0535,E2 19.7872} C_DIS
LIN {X 36.4034,Y 95.074,Z 100,A 63.766,B 24.9212,C -2.0503,E1 25.0585,E2 21.6771} C_DIS
LIN {X 39.2926,Y 93.9164,Z 100,A 61.9804,B 24.9214,C -2.0472,E1 25.0631,E2 23.4659} C_DIS
LIN {X 42.1993,Y 92.6473,Z 100,A 60.0097,B 24.9221,C -2.038,E1 25.0682,E2 25.4534} C_DIS
LIN {X 44.9041,Y 91.3667,Z 100,A 58.5066,B 24.9217,C -2.0429,E1 25.0719,E2 26.941} C_DIS
LIN {X 47.9568,Y 89.8032,Z 100,A 55.8357,B 24.9241,C -2.0119,E1 25.0787,E2 29.6776} C_DIS
LIN {X 51.9057,Y 87.5782,Z 100,A 54.2971,B 24.9214,C -2.0473,E1 25.0822,E2 31.128} C_DIS
LIN {X 54.209,Y 86.172,Z 100,A 52.6213,B 24.9221,C -2.0388,E1 25.0862,E2 32.8185} C_DIS
LIN {X 57.106,Y 84.2795,Z 100,A 50.602,B 24.9225,C -2.0329,E1 25.0909,E2 34.8451} C_DIS
LIN {X 59.9542,Y 82.2781,Z 100,A 47.2698,B 24.9268,C -1.9765,E1 25.0987,E2 38.2988} C_DIS
LIN {X 65.492,Y 77.9439,Z 100,A 44.8154,B 24.9229,C -2.0273,E1 25.1037,E2 40.6238} C_DIS
LIN {X 67.5456,Y 76.1705,Z 100,A 43.163,B 24.9235,C -2.0193,E1 25.1072,E2 42.2885} C_DIS
LIN {X 71.0929,Y 72.8719,Z 100,A 40.5752,B 24.9235,C -2.0191,E1 25.1124,E2 44.8661} C_DIS
LIN {X 73.0524,Y 70.9056,Z 100,A 38.806,B 24.9244,C -2.0076,E1 25.1159,E2 46.655} C_DIS
LIN {X 76.7198,Y 66.9194,Z 100,A 36.0353,B 24.9241,C -2.0118,E1 25.1211,E2 49.4036} C_DIS
LIN {X 78.474,Y 64.854,Z 100,A 34.4325,B 24.9246,C -2.0051,E1 25.124,E2 51.0147} C_DIS
LIN {X 80.4818,Y 62.3449,Z 100,A 32.5831,B 24.9251,C -1.9991,E1 25.1272,E2 52.8697} C_DIS
LIN {X 82.3958,Y 59.7935,Z 100,A 29.9271,B 24.9279,C -1.9605,E1 25.1317,E2 55.6039} C_DIS
LIN {X 85.2102,Y 55.7092,Z 100,A 28.4943,B 24.9244,C -2.0075,E1 25.1337,E2 56.9186} C_DIS
LIN {X 87.1188,Y 52.6736,Z 100,A 25.8969,B 24.9266,C -1.9789,E1 25.1376,E2 59.5704} C_DIS
LIN {X 88.9619,Y 49.4969,Z 100,A 23.7293,B 24.9273,C -1.9693,E1 25.1406,E2 61.7495} C_DIS
LIN {X 90.5902,Y 46.4496,Z 100,A 22.0123,B 24.927,C -1.9731,E1 25.1428,E2 63.4485} C_DIS
LIN {X 92.1173,Y 43.3441,Z 100,A 19.4505,B 24.9292,C -1.9429,E1 25.146,E2 66.0677} C_DIS
LIN {X 93.7617,Y 39.6598,Z 100,A 17.9619,B 24.9274,C -1.9678,E1 25.1475,E2 67.4893} C_DIS
LIN {X 94.7579,Y 37.2166,Z 100,A 16.3733,B 24.928,C -1.9593,E1 25.1492,E2 69.0893} C_DIS
LIN {X 95.8884,Y 34.2028,Z 100,A 14.5382,B 24.9285,C -1.953,E1 25.151,E2 70.929} C_DIS
LIN {X 96.8597,Y 31.3421,Z 100,A 12.9003,B 24.9287,C -1.9504,E1 25.1524,E2 72.5636} C_DIS
LIN {X 98.3597,Y 26.2602,Z 100,A 9.9215,B 24.9293,C -1.9415,E1 25.1547,E2 75.5465} C_DIS
LIN {X 99.1995,Y 22.8824,Z 100,A 8.0188,B 24.9296,C -1.9377,E1 25.1559,E2 77.4471} C_DIS
LIN {X 99.7648,Y 20.2771,Z 100,A 6.3682,B 24.9304,C -1.927,E1 25.1569,E2 79.1135} C_DIS
LIN {X 100.6478,Y 15.3039,Z 100,A 3.6134,B 24.9308,C -1.9216,E1 25.1582,E2 81.8648} C_DIS
LIN {X 101.1236,Y 11.7541,Z 100,A 1.5375,B 24.9314,C -1.9127,E1 25.1589,E2 83.9493} C_DIS
LIN {X 101.4791,Y 8.1314,Z 100,A -0.358,B 24.9314,C -1.9125,E1 25.1594,E2 85.8342} C_DIS
LIN {X 101.7013,Y 4.5864,Z 100,A -2.4504,B 24.9322,C -1.9022,E1 25.1597,E2 87.9383} C_DIS
LIN {X 101.7935,Y 1.53,Z 100,A -4.0307,B 24.9322,C -1.9024,E1 25.1597,E2 89.5088} C_DIS
LIN {X 101.7861,Y -1.9334,Z 100,A -5.9895,B 24.9326,C -1.8958,E1 25.1597,E2 91.4716} C_DIS
LIN {X 101.6572,Y -5.4752,Z 100,A -8.0737,B 24.9333,C -1.8856,E1 25.1595,E2 93.5673} C_DIS
LIN {X 101.4141,Y -8.917,Z 100,A -10.039,B 24.9339,C -1.8784,E1 25.159,E2 95.5381} C_DIS
LIN {X 101.0196,Y -12.6246,Z 100,A -12.064,B 24.9341,C -1.8746,E1 25.1584,E2 97.56} C_DIS
LIN {X 100.5505,Y -15.9337,Z 100,A -14.14,B 24.9351,C -1.8606,E1 25.1575,E2 99.6568} C_DIS
LIN {X 99.9753,Y -19.2113,Z 100,A -15.7852,B 24.9349,C -1.8639,E1 25.1567,E2 101.2846} C_DIS
LIN {X 98.8403,Y -24.3884,Z 100,A -18.3444,B 24.9343,C -1.8717,E1 25.1551,E2 103.8105} C_DIS
LIN {X 98.2727,Y -26.5823,Z 100,A -19.9672,B 24.9356,C -1.8534,E1 25.154,E2 105.4672} C_DIS
LIN {X 97.2816,Y -30.0073,Z 100,A -22.6933,B 24.9381,C -1.8178,E1 25.1517,E2 108.2616} C_DIS
LIN {X 95.8608,Y -34.2812,Z 100,A -24.5504,B 24.9367,C -1.8374,E1 25.15,E2 110.0622} C_DIS
LIN {X 94.6448,Y -37.5046,Z 100,A -26.3507,B 24.9367,C -1.8371,E1 25.1482,E2 111.8532} C_DIS
LIN {X 92.9542,Y -41.5182,Z 100,A -28.6717,B 24.9369,C -1.8349,E1 25.1457,E2 114.1665} C_DIS
LIN {X 91.8026,Y -44.0048,Z 100,A -30.374,B 24.9377,C -1.8237,E1 25.1436,E2 115.8861} C_DIS
LIN {X 90.2603,Y -47.0889,Z 100,A -32.3325,B 24.9381,C -1.8172,E1 25.1411,E2 117.8495} C_DIS
LIN {X 88.0435,Y -51.1144,Z 100,A -34.7821,B 24.9382,C -1.8152,E1 25.1378,E2 120.2911} C_DIS
LIN {X 86.6595,Y -53.4286,Z 100,A -36.4364,B 24.9389,C -1.8053,E1 25.1354,E2 121.9605} C_DIS
LIN {X 84.9749,Y -56.0661,Z 100,A -38.1018,B 24.9389,C -1.8042,E1 25.1329,E2 123.62} C_DIS
LIN {X 83.1895,Y -58.6851,Z 100,A -40.1038,B 24.9399,C -1.7904,E1 25.1296,E2 125.6447} C_DIS
LIN {X 80.5926,Y -62.2011,Z 100,A -42.3609,B 24.9399,C -1.792,E1 25.1259,E2 127.8874} C_DIS
LIN {X 78.1935,Y -65.1916,Z 100,A -44.4735,B 24.9401,C -1.7881,E1 25.1222,E2 129.9993} C_DIS
LIN {X 75.8733,Y -67.8776,Z 100,A -46.483,B 24.9405,C -1.7825,E1 25.1184,E2 132.0131} C_DIS
LIN {X 73.5572,Y -70.3819,Z 100,A -48.4245,B 24.9408,C -1.7768,E1 25.1147,E2 133.9596} C_DIS
LIN {X 71.2724,Y -72.6947,Z 100,A -50.2762,B 24.9412,C -1.7714,E1 25.1111,E2 135.8161} C_DIS
LIN {X 68.8001,Y -75.0379,Z 100,A -52.119,B 24.9412,C -1.7699,E1 25.1073,E2 137.655} C_DIS
LIN {X 66.1141,Y -77.415,Z 100,A -54.1132,B 24.9415,C -1.7662,E1 25.1031,E2 139.65} C_DIS
LIN {X 63.5483,Y -79.5364,Z 100,A -56.1229,B 24.9422,C -1.7566,E1 25.0987,E2 141.6747} C_DIS
LIN {X 60.5205,Y -81.8635,Z 100,A -57.9667,B 24.9417,C -1.7643,E1 25.0947,E2 143.4939} C_DIS
LIN {X 57.8327,Y -83.7832,Z 100,A -59.8719,B 24.942,C -1.7586,E1 25.0903,E2 145.4058} C_DIS
LIN {X 55.6692,Y -85.2366,Z 100,A -61.4589,B 24.9425,C -1.7509,E1 25.0866,E2 147.0057} C_DIS
LIN {X 52.9117,Y -86.9741,Z 100,A -63.2485,B 24.9427,C -1.7492,E1 25.0823,E2 148.7936} C_DIS
LIN {X 50.2647,Y -88.5318,Z 100,A -65.0349,B 24.943,C -1.7438,E1 25.078,E2 150.5875} C_DIS
LIN {X 47.236,Y -90.1829,Z 100,A -66.9579,B 24.9432,C -1.7412,E1 25.0733,E2 152.5111} C_DIS
LIN {X 44.2497,Y -91.6849,Z 100,A -68.7889,B 24.9432,C -1.7401,E1 25.0687,E2 154.3399} C_DIS
LIN {X 41.0681,Y -93.1543,Z 100,A -70.8113,B 24.9436,C -1.7351,E1 25.0635,E2 156.3691} C_DIS
LIN {X 37.7365,Y -94.5537,Z 100,A -73.2608,B 24.9448,C -1.7159,E1 25.0571,E2 158.8584} C_DIS
LIN {X 34.6302,Y -95.7338,Z 100,A -74.4615,B 24.9433,C -1.7396,E1 25.0541,E2 160.0006} C_DIS
LIN {X 32.3843,Y -96.5164,Z 100,A -76.0241,B 24.944,C -1.7291,E1 25.0499,E2 161.5848} C_DIS
LIN {X 27.8435,Y -97.9228,Z 100,A -78.6868,B 24.9441,C -1.7265,E1 25.0428,E2 164.2489} C_DIS
LIN {X 24.431,Y -98.8299,Z 100,A -80.6914,B 24.9443,C -1.7238,E1 25.0373,E2 166.257} C_DIS
LIN {X 20.9425,Y -99.6282,Z 100,A -82.9744,B 24.9451,C -1.7116,E1 25.031,E2 168.5658} C_DIS
LIN {X 16.9492,Y -100.3837,Z 100,A -84.9667,B 24.9445,C -1.7211,E1 25.0256,E2 170.5334} C_DIS
LIN {X 12.7789,Y -100.9996,Z 100,A -87.2396,B 24.9443,C -1.7233,E1 25.0194,E2 172.799} C_DIS
LIN {X 9.4778,Y -101.3623,Z 100,A -89.1758,B 24.9446,C -1.7197,E1 25.014,E2 174.7425} C_DIS
LIN {X 5.9727,Y -101.6297,Z 100,A -91.2575,B 24.9449,C -1.7149,E1 25.0081,E2 176.8348} C_DIS
LIN {X 2.8528,Y -101.7648,Z 100,A -92.8601,B 24.9445,C -1.7202,E1 25.0037,E2 178.4244} C_DIS
LIN {X 0.7106,Y -101.8004,Z 100,A -93.8591,B 24.9441,C -1.7278,E1 25.001,E2 179.4053} C_DIS
Enddeposition()
LIN {X 0.7106,Y -101.8004,Z 100,A -93.8591,B 24.9441,C -1.7278,E1 25.001,E2 179.4053} C_DIS
Startdeposition()
$VEL.CP = VEL_PRINT
LIN {X 1.649,Y -100.9132,Z 100,A -93.074,B 24.9424,C -1.7528,E1 25.0033,E2 178.561} C_DIS
LIN {X 4.7253,Y -100.8166,Z 100,A -90.7473,B 24.9409,C -1.7756,E1 25.01,E2 176.1808} C_DIS
LIN {X 9.2341,Y -100.5032,Z 100,A -88.438,B 24.9415,C -1.767,E1 25.0163,E2 173.8931} C_DIS
LIN {X 12.7051,Y -100.1239,Z 100,A -85.8003,B 24.9397,C -1.7937,E1 25.0238,E2 171.1943} C_DIS
LIN {X 16.9452,Y -99.4942,Z 100,A -84.1507,B 24.9416,C -1.765,E1 25.0282,E2 169.6143} C_DIS
LIN {X 24.1025,Y -98.0064,Z 100,A -80.0494,B 24.9415,C -1.7667,E1 25.0394,E2 165.5142} C_DIS
LIN {X 30.6513,Y -96.1605,Z 100,A -75.99,B 24.9407,C -1.7787,E1 25.0503,E2 161.4335} C_DIS
LIN {X 34.1501,Y -94.9744,Z 100,A -74.1548,B 24.9412,C -1.7711,E1 25.0551,E2 159.6199} C_DIS
LIN {X 37.6898,Y -93.6258,Z 100,A -71.3457,B 24.9393,C -1.8001,E1 25.0625,E2 156.7484} C_DIS
LIN {X 40.9451,Y -92.2495,Z 100,A -69.7278,B 24.9401,C -1.7877,E1 25.0666,E2 155.1638} C_DIS
LIN {X 43.9439,Y -90.8579,Z 100,A -67.4356,B 24.9388,C -1.8073,E1 25.0725,E2 152.8313} C_DIS
LIN {X 47.1819,Y -89.2191,Z 100,A -65.8297,B 24.9398,C -1.7926,E1 25.0763,E2 151.2646} C_DIS
LIN {X 50.4171,Y -87.4316,Z 100,A -63.8346,B 24.9398,C -1.7922,E1 25.0812,E2 149.2762} C_DIS
LIN {X 53.2642,Y -85.7271,Z 100,A -62.0146,B 24.9398,C -1.7932,E1 25.0855,E2 147.4596} C_DIS
LIN {X 55.8059,Y -84.0948,Z 100,A -60.4021,B 24.9398,C -1.7925,E1 25.0893,E2 145.8541} C_DIS
LIN {X 59.2882,Y -81.6777,Z 100,A -57.911,B 24.9392,C -1.8008,E1 25.095,E2 143.352} C_DIS
LIN {X 61.5739,Y -79.9675,Z 100,A -56.2257,B 24.9388,C -1.8068,E1 25.0987,E2 141.6586} C_DIS
LIN {X 64.4208,Y -77.6925,Z 100,A -54.1281,B 24.9384,C -1.8126,E1 25.1033,E2 139.5554} C_DIS
LIN {X 67.2358,Y -75.2696,Z 100,A -52.0541,B 24.9382,C -1.816,E1 25.1077,E2 137.4814} C_DIS
LIN {X 69.8114,Y -72.8877,Z 100,A -50.1203,B 24.938,C -1.8184,E1 25.1116,E2 135.5499} C_DIS
LIN {X 71.8377,Y -70.8907,Z 100,A -48.4667,B 24.9376,C -1.8239,E1 25.1149,E2 133.8903} C_DIS
LIN {X 74.3933,Y -68.204,Z 100,A -46.3749,B 24.9373,C -1.8287,E1 25.1189,E2 131.7964} C_DIS
LIN {X 76.8085,Y -65.4722,Z 100,A -44.3544,B 24.9371,C -1.832,E1 25.1226,E2 129.7772} C_DIS
LIN {X 79.0556,Y -62.7408,Z 100,A -42.3183,B 24.9366,C -1.8385,E1 25.1261,E2 127.7352} C_DIS
LIN {X 81.308,Y -59.7931,Z 100,A -40.5459,B 24.9372,C -1.8306,E1 25.1291,E2 125.9898} C_DIS
LIN {X 83.1573,Y -57.195,Z 100,A -38.3868,B 24.9359,C -1.8498,E1 25.1326,E2 123.796} C_DIS
LIN {X 85.0203,Y -54.385,Z 100,A -36.5729,B 24.9358,C -1.8511,E1 25.1354,E2 121.988} C_DIS
LIN {X 86.5214,Y -51.9661,Z 100,A -34.7221,B 24.9348,C -1.8654,E1 25.1381,E2 120.1131} C_DIS
LIN {X 89.2792,Y -47.0678,Z 100,A -31.1676,B 24.9331,C -1.8898,E1 25.1429,E2 116.5196} C_DIS
LIN {X 91.0311,Y -43.5834,Z 100,A -30.0485,B 24.9357,C -1.8514,E1 25.1441,E2 115.4971} C_DIS
LIN {X 93.3446,Y -38.3804,Z 100,A -26.325,B 24.9337,C -1.8812,E1 25.1484,E2 111.7235} C_DIS
LIN {X 94.6181,Y -35.1268,Z 100,A -24.4757,B 24.9337,C -1.8818,E1 25.1502,E2 109.8831} C_DIS
LIN {X 95.9295,Y -31.3651,Z 100,A -21.2543,B 24.9303,C -1.9286,E1 25.1531,E2 106.5694} C_DIS
LIN {X 97.3638,Y -26.5802,Z 100,A -19.2946,B 24.9322,C -1.9013,E1 25.1545,E2 104.6856} C_DIS
LIN {X 98.2766,Y -22.9758,Z 100,A -16.7537,B 24.9305,C -1.9258,E1 25.1562,E2 102.1016} C_DIS
LIN {X 99.0093,Y -19.5848,Z 100,A -15.4127,B 24.9319,C -1.9061,E1 25.1569,E2 100.8147} C_DIS
LIN {X 99.8792,Y -14.5049,Z 100,A -12.328,B 24.9307,C -1.922,E1 25.1583,E2 97.7106} C_DIS
LIN {X 100.2497,Y -11.6682,Z 100,A -10.3364,B 24.9293,C -1.9425,E1 25.159,E2 95.6826} C_DIS
LIN {X 100.5727,Y -8.4531,Z 100,A -8.7641,B 24.9296,C -1.9375,E1 25.1594,E2 94.1312} C_DIS
LIN {X 100.8343,Y -4.312,Z 100,A -6.5581,B 24.9296,C -1.939,E1 25.1597,E2 91.9349} C_DIS
LIN {X 100.9249,Y -0.5826,Z 100,A -4.6079,B 24.9296,C -1.939,E1 25.1597,E2 89.9964} C_DIS
LIN {X 100.8919,Y 2.6742,Z 100,A -2.4609,B 24.9282,C -1.9571,E1 25.1597,E2 87.8193} C_DIS
LIN {X 100.7084,Y 6.6335,Z 100,A -0.43,B 24.9283,C -1.9553,E1 25.1594,E2 85.8046} C_DIS
LIN {X 100.4163,Y 10.1421,Z 100,A 1.3516,B 24.9285,C -1.9528,E1 25.1589,E2 84.0396} C_DIS
LIN {X 99.9776,Y 13.8123,Z 100,A 3.5375,B 24.9278,C -1.963,E1 25.1582,E2 81.8425} C_DIS
LIN {X 98.8055,Y 20.5843,Z 100,A 6.969,B 24.9283,C -1.956,E1 25.1566,E2 78.4476} C_DIS
LIN {X 98.092,Y 23.7519,Z 100,A 9.6649,B 24.9253,C -1.9965,E1 25.1548,E2 75.6718} C_DIS
LIN {X 96.5653,Y 29.3532,Z 100,A 12.6731,B 24.9253,C -1.9947,E1 25.1525,E2 72.6851} C_DIS
LIN {X 95.5164,Y 32.6023,Z 100,A 14.6795,B 24.9247,C -2.0033,E1 25.1507,E2 70.6697} C_DIS
LIN {X 94.2864,Y 36.0043,Z 100,A 16.6121,B 24.9247,C -2.0044,E1 25.1488,E2 68.7453} C_DIS
LIN {X 92.6511,Y 40.0254,Z 100,A 20.0757,B 24.921,C -2.0525,E1 25.1449,E2 65.1872} C_DIS
LIN {X 90.3194,Y 45.0401,Z 100,A 22.1705,B 24.9236,C -2.0185,E1 25.1425,E2 63.1838} C_DIS
LIN {X 87.9651,Y 49.4812,Z 100,A 25.1066,B 24.9228,C -2.0297,E1 25.1386,E2 60.2369} C_DIS
LIN {X 86.2033,Y 52.4895,Z 100,A 26.8143,B 24.9232,C -2.024,E1 25.1362,E2 58.5513} C_DIS
LIN {X 84.5711,Y 55.0837,Z 100,A 28.5907,B 24.9227,C -2.03,E1 25.1335,E2 56.7698} C_DIS
LIN {X 82.2698,Y 58.4625,Z 100,A 31.1405,B 24.9216,C -2.0451,E1 25.1294,E2 54.1968} C_DIS
LIN {X 80.0202,Y 61.5056,Z 100,A 33.0757,B 24.9218,C -2.0418,E1 25.1262,E2 52.2786} C_DIS
LIN {X 78.1291,Y 63.8921,Z 100,A 34.9312,B 24.9211,C -2.051,E1 25.1229,E2 50.41} C_DIS
LIN {X 76.1388,Y 66.25,Z 100,A 36.9988,B 24.9198,C -2.0677,E1 25.1191,E2 48.3123} C_DIS
LIN {X 73.0967,Y 69.5945,Z 100,A 39.2589,B 24.9203,C -2.0611,E1 25.1148,E2 46.0777} C_DIS
LIN {X 70.4736,Y 72.2495,Z 100,A 41.4783,B 24.9197,C -2.0696,E1 25.1104,E2 43.8476} C_DIS
LIN {X 67.479,Y 75.0519,Z 100,A 43.6284,B 24.9199,C -2.0672,E1 25.106,E2 41.7117} C_DIS
LIN {X 64.8726,Y 77.3171,Z 100,A 46.648,B 24.9162,C -2.1132,E1 25.0993,E2 38.595} C_DIS
LIN {X 60.3452,Y 80.8986,Z 100,A 49.0414,B 24.9186,C -2.0839,E1 25.0942,E2 36.2797} C_DIS
LIN {X 56.7373,Y 83.4689,Z 100,A 51.2997,B 24.919,C -2.078,E1 25.089,E2 34.0431} C_DIS
LIN {X 53.982,Y 85.2787,Z 100,A 53.3995,B 24.9181,C -2.0898,E1 25.084,E2 31.9221} C_DIS
LIN {X 51.0211,Y 87.0813,Z 100,A 55.5449,B 24.9173,C -2.0997,E1 25.0788,E2 29.7599} C_DIS
LIN {X 45.6566,Y 90.0096,Z 100,A 58.7011,B 24.9179,C -2.0921,E1 25.0711,E2 26.6306} C_DIS
LIN {X 43.4456,Y 91.0973,Z 100,A 60.1912,B 24.9175,C -2.0973,E1 25.0673,E2 25.1321} C_DIS
LIN {X 39.6668,Y 92.806,Z 100,A 62.4148,B 24.9177,C -2.0949,E1 25.0617,E2 22.9197} C_DIS
LIN {X 36.3273,Y 94.164,Z 100,A 64.5032,B 24.9174,C -2.0985,E1 25.0563,E2 20.8273} C_DIS
LIN {X 33.1706,Y 95.3201,Z 100,A 66.4125,B 24.9173,C -2.1003,E1 25.0512,E2 18.9177} C_DIS
LIN {X 28.9885,Y 96.6742,Z 100,A 68.8635,B 24.9173,C -2.1005,E1 25.0447,E2 16.4707} C_DIS
LIN {X 26.5173,Y 97.3808,Z 100,A 70.4647,B 24.9168,C -2.1069,E1 25.0404,E2 14.8569} C_DIS
LIN {X 19.6616,Y 98.9942,Z 100,A 74.1397,B 24.9176,C -2.0966,E1 25.0304,E2 11.2112} C_DIS
LIN {X 14.6841,Y 99.8538,Z 100,A 77.1544,B 24.9171,C -2.1031,E1 25.0221,E2 8.1842} C_DIS
LIN {X 9.9778,Y 100.4335,Z 100,A 79.9216,B 24.9168,C -2.1064,E1 25.0144,E2 5.4112} C_DIS
LIN {X 6.2845,Y 100.732,Z 100,A 81.7764,B 24.9175,C -2.0971,E1 25.0093,E2 3.5791} C_DIS
LIN {X 3.25,Y 100.8743,Z 100,A 84.0017,B 24.916,C -2.1157,E1 25.003,E2 1.3103} C_DIS
LIN {X -1.5091,Y 100.9158,Z 100,A 86.3509,B 24.9171,C -2.102,E1 24.9965,E2 -1.0063} C_DIS
LIN {X -4.8669,Y 100.8105,Z 100,A 88.7288,B 24.9158,C -2.1188,E1 24.9898,E2 -3.4247} C_DIS
LIN {X -8.2544,Y 100.5886,Z 100,A 90.1755,B 24.9173,C -2.1002,E1 24.9858,E2 -4.8278} C_DIS
LIN {X -14.276,Y 99.9117,Z 100,A 93.3968,B 24.9181,C -2.0902,E1 24.977,E2 -8.0274} C_DIS
LIN {X -21.542,Y 98.6007,Z 100,A 98.7617,B 24.9149,C -2.1298,E1 24.962,E2 -13.4924} C_DIS
LIN {X -26.632,Y 97.3498,Z 100,A 100.8224,B 24.9178,C -2.0932,E1 24.9567,E2 -15.4693} C_DIS
LIN {X -30.4865,Y 96.2135,Z 100,A 103.1591,B 24.9178,C -2.0927,E1 24.9504,E2 -17.8087} C_DIS
LIN {X -33.7488,Y 95.1173,Z 100,A 105.0902,B 24.9181,C -2.0894,E1 24.9453,E2 -19.7358} C_DIS
LIN {X -36.9106,Y 93.9349,Z 100,A 107.3641,B 24.9173,C -2.0998,E1 24.9393,E2 -22.0391} C_DIS
LIN {X -41.2029,Y 92.1334,Z 100,A 109.6545,B 24.9186,C -2.0832,E1 24.9336,E2 -24.2956} C_DIS
LIN {X -45.6422,Y 90.0169,Z 100,A 112.3339,B 24.9193,C -2.0748,E1 24.9269,E2 -26.9618} C_DIS
LIN {X -49.7601,Y 87.8091,Z 100,A 115.1278,B 24.9193,C -2.0752,E1 24.92,E2 -29.7647} C_DIS
LIN {X -52.4393,Y 86.2338,Z 100,A 116.8567,B 24.9196,C -2.0708,E1 24.9159,E2 -31.4883} C_DIS
LIN {X -55.8399,Y 84.0725,Z 100,A 119.5211,B 24.9189,C -2.0797,E1 24.9096,E2 -34.1827} C_DIS
LIN {X -60.209,Y 81.0017,Z 100,A 122.2383,B 24.9202,C -2.0624,E1 24.9035,E2 -36.8682} C_DIS
LIN {X -62.7408,Y 79.0556,Z 100,A 124.0855,B 24.9204,C -2.0597,E1 24.8994,E2 -38.7158} C_DIS
LIN {X -65.7469,Y 76.5744,Z 100,A 126.3883,B 24.9206,C -2.058,E1 24.8945,E2 -41.0232} C_DIS
LIN {X -68.7054,Y 73.9323,Z 100,A 128.5691,B 24.9212,C -2.0503,E1 24.89,E2 -43.1945} C_DIS
LIN {X -71.1248,Y 71.6065,Z 100,A 130.3912,B 24.9217,C -2.0428,E1 24.8864,E2 -45.0065} C_DIS
LIN {X -73.4071,Y 69.2645,Z 100,A 131.9842,B 24.9228,C -2.0291,E1 24.8834,E2 -46.5737} C_DIS
LIN {X -75.3221,Y 67.1771,Z 100,A 134.1969,B 24.9215,C -2.0461,E1 24.8791,E2 -48.8366} C_DIS
LIN {X -78.3443,Y 63.6265,Z 100,A 136.5972,B 24.9227,C -2.0306,E1 24.8749,E2 -51.2112} C_DIS
LIN {X -80.5902,Y 60.7569,Z 100,A 139.0155,B 24.9222,C -2.0372,E1 24.8707,E2 -53.6567} C_DIS
LIN {X -83.8944,Y 56.1065,Z 100,A 142.3888,B 24.9225,C -2.0329,E1 24.8654,E2 -57.0365} C_DIS
LIN {X -85.7669,Y 53.2005,Z 100,A 143.9147,B 24.9241,C -2.0122,E1 24.8632,E2 -58.5209} C_DIS
LIN {X -89.7418,Y 46.1805,Z 100,A 148.5227,B 24.925,C -1.9998,E1 24.857,E2 -63.1234} C_DIS
LIN {X -91.2527,Y 43.1212,Z 100,A 150.3273,B 24.9258,C -1.9894,E1 24.8548,E2 -64.9131} C_DIS
LIN {X -92.8748,Y 39.5037,Z 100,A 152.7511,B 24.9258,C -1.9886,E1 24.8521,E2 -67.3481} C_DIS
LIN {X -94.1713,Y 36.3074,Z 100,A 154.7308,B 24.9263,C -1.9833,E1 24.85,E2 -69.3263} C_DIS
LIN {X -95.3074,Y 33.207,Z 100,A 156.6803,B 24.9265,C -1.9801,E1 24.8482,E2 -71.2792} C_DIS
LIN {X -96.8589,Y 28.3661,Z 100,A 159.4628,B 24.9274,C -1.9675,E1 24.8459,E2 -74.0476} C_DIS
LIN {X -97.9501,Y 24.3333,Z 100,A 161.9103,B 24.9278,C -1.9625,E1 24.8442,E2 -76.4976} C_DIS
LIN {X -98.7269,Y 20.9634,Z 100,A 163.9264,B 24.9281,C -1.9581,E1 24.843,E2 -78.5149} C_DIS
LIN {X -99.4249,Y 17.3524,Z 100,A 165.8555,B 24.929,C -1.946,E1 24.842,E2 -80.4266} C_DIS
LIN {X -100.0146,Y 13.5488,Z 100,A 168.1242,B 24.9293,C -1.9418,E1 24.8411,E2 -82.6988} C_DIS
LIN {X -100.47,Y 9.593,Z 100,A 171.0884,B 24.9281,C -1.9587,E1 24.8402,E2 -85.7211} C_DIS
LIN {X -100.7785,Y 5.4647,Z 100,A 172.9091,B 24.93,C -1.9329,E1 24.8399,E2 -87.4912} C_DIS
LIN {X -100.8919,Y 2.6743,Z 100,A 175.1799,B 24.9286,C -1.9514,E1 24.8399,E2 -89.8197} C_DIS
LIN {X -100.9079,Y -1.937,Z 100,A 177.5658,B 24.9298,C -1.9349,E1 24.8399,E2 -92.1808} C_DIS
LIN {X -100.7695,Y -5.6272,Z 100,A 179.1086,B 24.9317,C -1.9092,E1 24.8401,E2 -93.6715} C_DIS
LIN {X -100.0749,Y -13.0837,Z 100,A -176.8136,B 24.9331,C -1.8896,E1 24.8413,E2 -97.7271} C_DIS
LIN {X -99.6352,Y -16.1024,Z 100,A -174.7664,B 24.9327,C -1.8949,E1 24.8421,E2 -99.7992} C_DIS
LIN {X -99.0329,Y -19.4622,Z 100,A -172.8379,B 24.9331,C -1.8886,E1 24.8431,E2 -101.7239} C_DIS
LIN {X -98.309,Y -22.8365,Z 100,A -170.879,B 24.9336,C -1.8825,E1 24.8443,E2 -103.6798} C_DIS
LIN {X -97.45,Y -26.2614,Z 100,A -168.8712,B 24.934,C -1.8765,E1 24.8457,E2 -105.685} C_DIS
LIN {X -96.5931,Y -29.262,Z 100,A -166.462,B 24.9328,C -1.8932,E1 24.8477,E2 -108.1481} C_DIS
LIN {X -95.3384,Y -33.1185,Z 100,A -164.7734,B 24.9348,C -1.8651,E1 24.8492,E2 -109.7791} C_DIS
LIN {X -94.1409,Y -36.3862,Z 100,A -162.9455,B 24.9356,C -1.8541,E1 24.8509,E2 -111.5911} C_DIS
LIN {X -91.867,Y -41.7941,Z 100,A -159.3567,B 24.9356,C -1.8535,E1 24.8549,E2 -115.1983} C_DIS
LIN {X -90.2945,Y -45.0903,Z 100,A -157.4103,B 24.9363,C -1.8433,E1 24.8573,E2 -117.1309} C_DIS
LIN {X -88.7232,Y -48.1077,Z 100,A -155.4282,B 24.9366,C -1.8398,E1 24.8599,E2 -119.1151} C_DIS
LIN {X -87.1776,Y -50.8582,Z 100,A -153.2051,B 24.9358,C -1.8501,E1 24.8631,E2 -121.3743} C_DIS
LIN {X -84.9255,Y -54.5327,Z 100,A -150.9024,B 24.9366,C -1.8387,E1 24.8665,E2 -123.6615} C_DIS
LIN {X -82.3413,Y -58.3624,Z 100,A -148.2625,B 24.937,C -1.8326,E1 24.8707,E2 -126.3} C_DIS
LIN {X -79.9052,Y -61.6548,Z 100,A -146.1875,B 24.938,C -1.8182,E1 24.8741,E2 -128.3505} C_DIS
LIN {X -77.6877,Y -64.4265,Z 100,A -144.2157,B 24.9385,C -1.8119,E1 24.8776,E2 -130.3166} C_DIS
LIN {X -74.876,Y -67.6755,Z 100,A -141.6377,B 24.9385,C -1.8112,E1 24.8824,E2 -132.9046} C_DIS
LIN {X -72.4128,Y -70.3042,Z 100,A -139.6063,B 24.9388,C -1.8063,E1 24.8863,E2 -134.933} C_DIS
LIN {X -68.7501,Y -73.8909,Z 100,A -136.6588,B 24.9392,C -1.8016,E1 24.8922,E2 -137.8816} C_DIS
LIN {X -66.3066,Y -76.0895,Z 100,A -134.8214,B 24.9395,C -1.7969,E1 24.8961,E2 -139.7151} C_DIS
LIN {X -63.652,Y -78.3237,Z 100,A -132.4962,B 24.9389,C -1.806,E1 24.9011,E2 -142.0708} C_DIS
LIN {X -61.1325,Y -80.3077,Z 100,A -131.1559,B 24.9403,C -1.7855,E1 24.904,E2 -143.367} C_DIS
LIN {X -58.4487,Y -82.2797,Z 100,A -129.0482,B 24.9399,C -1.7901,E1 24.9088,E2 -145.4931} C_DIS
LIN {X -54.9842,Y -84.6357,Z 100,A -126.6688,B 24.9402,C -1.7863,E1 24.9143,E2 -147.8713} C_DIS
LIN {X -49.3348,Y -88.0469,Z 100,A -122.8743,B 24.9404,C -1.7826,E1 24.9235,E2 -151.6686} C_DIS
LIN {X -45.3256,Y -90.1776,Z 100,A -120.4615,B 24.9411,C -1.7733,E1 24.9294,E2 -154.0657} C_DIS
LIN {X -42.4276,Y -91.5755,Z 100,A -118.5004,B 24.9409,C -1.7761,E1 24.9344,E2 -156.0385} C_DIS
LIN {X -39.1301,Y -93.0322,Z 100,A -116.5735,B 24.9413,C -1.7695,E1 24.9393,E2 -157.9543} C_DIS
LIN {X -35.861,Y -94.3406,Z 100,A -114.5363,B 24.9413,C -1.769,E1 24.9446,E2 -159.9947} C_DIS
LIN {X -31.7999,Y -95.7869,Z 100,A -112.0157,B 24.9413,C -1.7697,E1 24.9513,E2 -162.5216} C_DIS
LIN {X -27.2615,Y -97.1753,Z 100,A -108.5424,B 24.9395,C -1.7971,E1 24.9608,E2 -166.0656} C_DIS
LIN {X -22.5447,Y -98.3764,Z 100,A -106.82,B 24.9422,C -1.7565,E1 24.9652,E2 -167.694} C_DIS
LIN {X -17.8561,Y -99.3344,Z 100,A -103.9325,B 24.9418,C -1.7618,E1 24.9732,E2 -170.5973} C_DIS
LIN {X -13.4904,Y -100.0221,Z 100,A -101.3237,B 24.9416,C -1.7649,E1 24.9804,E2 -173.2157} C_DIS
LIN {X -10.2214,Y -100.408,Z 100,A -99.4506,B 24.9416,C -1.7649,E1 24.9856,E2 -175.0899} C_DIS
LIN {X -6.2713,Y -100.7324,Z 100,A -97.068,B 24.9413,C -1.7699,E1 24.9923,E2 -177.4853} C_DIS
LIN {X -2.204,Y -100.903,Z 100,A -94.881,B 24.9416,C -1.7655,E1 24.9984,E2 -179.6621} C_DIS
LIN {X 0.7043,Y -100.9199,Z 100,A -93.729,B 24.9428,C -1.7469,E1 25.0015,E2 -180.7702} C_DIS
Enddeposition()
LIN {X 0.7043,Y -100.9199,Z 100,A -93.729,B 24.9428,C -1.7469,E1 25.0015,E2 -180.7702} C_DIS
Startdeposition()
$VEL.CP = VEL_PRINT
LIN {X 0.2437,Y -100.0489,Z 100,A -94.4606,B 24.943,C -1.7446,E1 24.9994,E2 -180.033} C_DIS
LIN {X -3.186,Y -99.9979,Z 100,A -96.6363,B 24.9435,C -1.7365,E1 24.9933,E2 -177.8379} C_DIS
LIN {X -8.5851,Y -99.6813,Z 100,A -99.6549,B 24.9433,C -1.7393,E1 24.9849,E2 -174.8249} C_DIS
LIN {X -12.3411,Y -99.2858,Z 100,A -102.1635,B 24.9441,C -1.727,E1 24.9778,E2 -172.2854} C_DIS
LIN {X -15.7439,Y -98.8031,Z 100,A -103.4813,B 24.9425,C -1.7513,E1 24.9744,E2 -171.0241} C_DIS
LIN {X -19.199,Y -98.1896,Z 100,A -105.5953,B 24.9427,C -1.7482,E1 24.9685,E2 -168.9005} C_DIS
LIN {X -21.8744,Y -97.6296,Z 100,A -107.7034,B 24.944,C -1.7292,E1 24.9627,E2 -166.7446} C_DIS
LIN {X -25.1227,Y -96.8432,Z 100,A -109.3848,B 24.9433,C -1.7387,E1 24.9582,E2 -165.0835} C_DIS
LIN {X -28.5084,Y -95.9009,Z 100,A -111.1358,B 24.9426,C -1.7495,E1 24.9535,E2 -163.3553} C_DIS
LIN {X -31.9534,Y -94.8087,Z 100,A -113.6585,B 24.9436,C -1.7349,E1 24.9467,E2 -160.7931} C_DIS
LIN {X -35.0471,Y -93.7101,Z 100,A -115.0038,B 24.9422,C -1.7557,E1 24.9433,E2 -159.4946} C_DIS
LIN {X -37.7232,Y -92.6643,Z 100,A -116.7479,B 24.9424,C -1.7538,E1 24.9388,E2 -157.7421} C_DIS
LIN {X -40.8184,Y -91.3437,Z 100,A -118.7887,B 24.9424,C -1.7518,E1 24.9335,E2 -155.6918} C_DIS
LIN {X -44.8281,Y -89.4447,Z 100,A -121.3579,B 24.9424,C -1.7538,E1 24.9271,E2 -153.1208} C_DIS
LIN {X -48.2029,Y -87.6728,Z 100,A -123.9442,B 24.9431,C -1.7425,E1 24.9206,E2 -150.5001} C_DIS
LIN {X -51.2372,Y -85.9338,Z 100,A -125.596,B 24.9421,C -1.7578,E1 24.9167,E2 -148.8796} C_DIS
LIN {X -54.5039,Y -83.9008,Z 100,A -127.8674,B 24.9421,C -1.7587,E1 24.9114,E2 -146.6033} C_DIS
LIN {X -57.3081,Y -82.0095,Z 100,A -129.8473,B 24.9419,C -1.7605,E1 24.9068,E2 -144.6207} C_DIS
LIN {X -60.6659,Y -79.5589,Z 100,A -132.7451,B 24.9428,C -1.7467,E1 24.9003,E2 -141.6798} C_DIS
LIN {X -64.1308,Y -76.792,Z 100,A -134.4091,B 24.9405,C -1.7818,E1 24.8969,E2 -140.0929} C_DIS
LIN {X -66.3091,Y -74.9209,Z 100,A -136.2602,B 24.9408,C -1.7778,E1 24.8929,E2 -138.225} C_DIS
LIN {X -70.6285,Y -70.8627,Z 100,A -139.4816,B 24.9399,C -1.7907,E1 24.8865,E2 -135.0212} C_DIS
LIN {X -72.6393,Y -68.7995,Z 100,A -141.311,B 24.9401,C -1.7881,E1 24.8829,E2 -133.1777} C_DIS
LIN {X -76.6891,Y -64.2547,Z 100,A -144.5468,B 24.939,C -1.8046,E1 24.877,E2 -129.9666} C_DIS
LIN {X -79.0118,Y -61.3759,Z 100,A -147.4182,B 24.9403,C -1.784,E1 24.8719,E2 -127.0325} C_DIS
LIN {X -81.1827,Y -58.4747,Z 100,A -148.7859,B 24.9384,C -1.8132,E1 24.8697,E2 -125.7278} C_DIS
LIN {X -83.9096,Y -54.4893,Z 100,A -151.8214,B 24.9385,C -1.811,E1 24.865,E2 -122.6719} C_DIS
LIN {X -86.5809,Y -50.1355,Z 100,A -154.5331,B 24.9375,C -1.826,E1 24.8611,E2 -119.982} C_DIS
LIN {X -87.9583,Y -47.6765,Z 100,A -156.3067,B 24.9375,C -1.8249,E1 24.8587,E2 -118.1966} C_DIS
LIN {X -89.5875,Y -44.54,Z 100,A -158.3411,B 24.9372,C -1.8302,E1 24.8561,E2 -116.1638} C_DIS
LIN {X -91.1218,Y -41.3107,Z 100,A -161.7573,B 24.9399,C -1.7905,E1 24.8521,E2 -112.6342} C_DIS
LIN {X -93.6674,Y -35.1599,Z 100,A -164.0693,B 24.9357,C -1.8514,E1 24.8498,E2 -110.4545} C_DIS
LIN {X -95.7583,Y -28.9891,Z 100,A -167.8807,B 24.9352,C -1.8598,E1 24.8465,E2 -106.6413} C_DIS
LIN {X -96.8585,Y -25.0631,Z 100,A -170.3584,B 24.935,C -1.8621,E1 24.8446,E2 -104.1548} C_DIS
LIN {X -97.5987,Y -22.0107,Z 100,A -172.2641,B 24.9349,C -1.8641,E1 24.8434,E2 -102.2426} C_DIS
LIN {X -98.3601,Y -18.3132,Z 100,A -174.3714,B 24.9343,C -1.8726,E1 24.8423,E2 -100.1432} C_DIS
LIN {X -98.9267,Y -14.9444,Z 100,A -176.4608,B 24.9341,C -1.8744,E1 24.8413,E2 -98.0456} C_DIS
LIN {X -99.7256,Y -8.0319,Z 100,A 179.6731,B 24.933,C -1.891,E1 24.8402,E2 -94.196} C_DIS
LIN {X -100.0283,Y -2.0232,Z 100,A 175.6367,B 24.9336,C -1.8825,E1 24.8398,E2 -90.115} C_DIS
LIN {X -100.0344,Y 1.6896,Z 100,A 174.119,B 24.9316,C -1.9094,E1 24.8398,E2 -88.6524} C_DIS
LIN {X -99.934,Y 4.8148,Z 100,A 171.516,B 24.9331,C -1.8884,E1 24.8402,E2 -85.9836} C_DIS
LIN {X -99.632,Y 9.1203,Z 100,A 169.7787,B 24.9308,C -1.9206,E1 24.8406,E2 -84.3126} C_DIS
LIN {X -99.311,Y 12.1362,Z 100,A 167.9299,B 24.9308,C -1.9224,E1 24.8412,E2 -82.4572} C_DIS
LIN {X -98.5668,Y 17.1639,Z 100,A 164.9827,B 24.9301,C -1.9306,E1 24.8424,E2 -79.5118} C_DIS
LIN {X -97.8816,Y 20.7185,Z 100,A 162.8961,B 24.9297,C -1.9367,E1 24.8436,E2 -77.4276} C_DIS
LIN {X -97.099,Y 24.1177,Z 100,A 160.5772,B 24.93,C -1.9325,E1 24.8451,E2 -75.085} C_DIS
LIN {X -95.9778,Y 28.2493,Z 100,A 157.7371,B 24.9304,C -1.9275,E1 24.8474,E2 -72.2165} C_DIS
LIN {X -94.5842,Y 32.6165,Z 100,A 156.0074,B 24.9276,C -1.9651,E1 24.8489,E2 -70.5668} C_DIS
LIN {X -93.5805,Y 35.3893,Z 100,A 154.1626,B 24.9276,C -1.9651,E1 24.8506,E2 -68.7117} C_DIS
LIN {X -91.4664,Y 40.5459,Z 100,A 150.9619,B 24.9269,C -1.9746,E1 24.8541,E2 -65.5156} C_DIS
LIN {X -90.4664,Y 42.7302,Z 100,A 149.5673,B 24.9266,C -1.9781,E1 24.8557,E2 -64.1218} C_DIS
LIN {X -89.0846,Y 45.5374,Z 100,A 147.2631,B 24.9275,C -1.9664,E1 24.8587,E2 -61.7774} C_DIS
LIN {X -87.4331,Y 48.633,Z 100,A 145.4386,B 24.9266,C -1.9784,E1 24.8611,E2 -59.9718} C_DIS
LIN {X -85.439,Y 52.0567,Z 100,A 143.1841,B 24.9261,C -1.9853,E1 24.8644,E2 -57.7223} C_DIS
LIN {X -82.1725,Y 57.0736,Z 100,A 139.358,B 24.9264,C -1.9817,E1 24.8704,E2 -53.8684} C_DIS
LIN {X -79.76,Y 60.4003,Z 100,A 137.9489,B 24.9235,C -2.0196,E1 24.8726,E2 -52.543} C_DIS
LIN {X -77.2987,Y 63.521,Z 100,A 134.8141,B 24.9252,C -1.9967,E1 24.8782,E2 -49.339} C_DIS
LIN {X -74.941,Y 66.2858,Z 100,A 132.8671,B 24.9245,C -2.0065,E1 24.8818,E2 -47.4066} C_DIS
LIN {X -71.6682,Y 69.8116,Z 100,A 130.4041,B 24.9233,C -2.0231,E1 24.8865,E2 -44.9725} C_DIS
LIN {X -69.0577,Y 72.3948,Z 100,A 128.0326,B 24.9236,C -2.0191,E1 24.8913,E2 -42.5815} C_DIS
LIN {X -64.3735,Y 76.5903,Z 100,A 124.6497,B 24.9224,C -2.0346,E1 24.8983,E2 -39.2223} C_DIS
LIN {X -61.8641,Y 78.6295,Z 100,A 122.9048,B 24.9218,C -2.0423,E1 24.9021,E2 -37.4892} C_DIS
LIN {X -58.2115,Y 81.3704,Z 100,A 119.5042,B 24.9234,C -2.021,E1 24.9099,E2 -34.0259} C_DIS
LIN {X -54.4533,Y 83.9332,Z 100,A 117.6891,B 24.921,C -2.0529,E1 24.914,E2 -32.2808} C_DIS
LIN {X -48.2102,Y 87.6684,Z 100,A 113.5849,B 24.9202,C -2.0625,E1 24.9239,E2 -28.1872} C_DIS
LIN {X -45.4384,Y 89.1352,Z 100,A 110.8084,B 24.9226,C -2.0318,E1 24.931,E2 -25.33} C_DIS
LIN {X -41.0618,Y 91.234,Z 100,A 108.6582,B 24.9206,C -2.0576,E1 24.9363,E2 -23.236} C_DIS
LIN {X -36.4114,Y 93.1878,Z 100,A 105.8993,B 24.9199,C -2.0662,E1 24.9434,E2 -20.4913} C_DIS
LIN {X -33.0084,Y 94.4467,Z 100,A 103.9329,B 24.9194,C -2.0727,E1 24.9485,E2 -18.5365} C_DIS
LIN {X -29.1371,Y 95.7132,Z 100,A 101.6101,B 24.9192,C -2.0758,E1 24.9547,E2 -16.2167} C_DIS
LIN {X -26.0823,Y 96.589,Z 100,A 99.0562,B 24.921,C -2.0519,E1 24.9617,E2 -13.6023} C_DIS
LIN {X -21.9548,Y 97.6117,Z 100,A 97.4425,B 24.9186,C -2.0831,E1 24.9659,E2 -12.0604} C_DIS
LIN {X -16.4758,Y 98.6826,Z 100,A 94.0946,B 24.9188,C -2.0802,E1 24.9751,E2 -8.7022} C_DIS
LIN {X -9.9144,Y 99.5574,Z 100,A 90.6044,B 24.9178,C -2.0932,E1 24.9847,E2 -5.2403} C_DIS
LIN {X -4.6899,Y 99.9393,Z 100,A 87.5082,B 24.918,C -2.091,E1 24.9934,E2 -2.1376} C_DIS
LIN {X -2.2257,Y 100.0245,Z 100,A 85.5523,B 24.9195,C -2.0718,E1 24.9989,E2 -0.1359} C_DIS
LIN {X 2.3457,Y 100.0217,Z 100,A 82.7653,B 24.92,C -2.0661,E1 25.0067,E2 2.6643} C_DIS
LIN {X 5.815,Y 99.8798,Z 100,A 81.3847,B 24.9182,C -2.0881,E1 25.0105,E2 3.992} C_DIS
LIN {X 8.6492,Y 99.6755,Z 100,A 79.0008,B 24.9204,C -2.0605,E1 25.0173,E2 6.4401} C_DIS
LIN {X 12.6149,Y 99.2504,Z 100,A 77.3366,B 24.9187,C -2.0826,E1 25.0217,E2 8.0507} C_DIS
LIN {X 17.1612,Y 98.5673,Z 100,A 74.8601,B 24.9183,C -2.0875,E1 25.0285,E2 10.5131} C_DIS
LIN {X 22.8656,Y 97.4012,Z 100,A 71.3408,B 24.9189,C -2.0791,E1 25.0382,E2 14.0478} C_DIS
LIN {X 25.4665,Y 96.7549,Z 100,A 69.8014,B 24.919,C -2.078,E1 25.0423,E2 15.5875} C_DIS
LIN {X 28.8262,Y 95.8066,Z 100,A 67.4061,B 24.9203,C -2.0619,E1 25.0488,E2 18.0169} C_DIS
LIN {X 31.9928,Y 94.7954,Z 100,A 66.0187,B 24.9189,C -2.0795,E1 25.0524,E2 19.3599} C_DIS
LIN {X 35.0059,Y 93.7257,Z 100,A 64.0629,B 24.9194,C -2.0732,E1 25.0576,E2 21.3266} C_DIS
LIN {X 38.3947,Y 92.3894,Z 100,A 61.9633,B 24.9196,C -2.0705,E1 25.063,E2 23.4277} C_DIS
LIN {X 40.9716,Y 91.2747,Z 100,A 60.5637,B 24.9191,C -2.0766,E1 25.0665,E2 24.8096} C_DIS
LIN {X 43.3665,Y 90.1613,Z 100,A 58.9259,B 24.9196,C -2.07,E1 25.0707,E2 26.4586} C_DIS
LIN {X 48.1918,Y 87.678,Z 100,A 55.6789,B 24.9204,C -2.0606,E1 25.0787,E2 29.7188} C_DIS
LIN {X 51.5059,Y 85.7738,Z 100,A 53.4638,B 24.9207,C -2.0564,E1 25.0841,E2 31.937} C_DIS
LIN {X 55.531,Y 83.2245,Z 100,A 50.8166,B 24.9207,C -2.0552,E1 25.0903,E2 34.5785} C_DIS
LIN {X 57.8731,Y 81.6119,Z 100,A 48.8087,B 24.9221,C -2.038,E1 25.0949,E2 36.62} C_DIS
LIN {X 60.7415,Y 79.4999,Z 100,A 46.5402,B 24.9231,C -2.0256,E1 25.1,E2 38.9095} C_DIS
LIN {X 64.2532,Y 76.6903,Z 100,A 44.6913,B 24.9213,C -2.0485,E1 25.1038,E2 40.6973} C_DIS
LIN {X 66.8951,Y 74.3963,Z 100,A 42.7667,B 24.9213,C -2.0476,E1 25.1079,E2 42.6163} C_DIS
LIN {X 69.8542,Y 71.6271,Z 100,A 40.3334,B 24.9221,C -2.0384,E1 25.1128,E2 45.0613} C_DIS
LIN {X 72.3215,Y 69.1338,Z 100,A 38.2099,B 24.9228,C -2.0296,E1 25.117,E2 47.1964} C_DIS
LIN {X 75.5578,Y 65.5806,Z 100,A 35.915,B 24.9219,C -2.0412,E1 25.1212,E2 49.4538} C_DIS
LIN {X 77.1036,Y 63.7558,Z 100,A 34.2991,B 24.9229,C -2.0284,E1 25.1241,E2 51.0926} C_DIS
LIN {X 79.4369,Y 60.8242,Z 100,A 32.1568,B 24.9232,C -2.0234,E1 25.1278,E2 53.2367} C_DIS
LIN {X 82.1425,Y 57.1167,Z 100,A 29.3658,B 24.9242,C -2.0104,E1 25.1324,E2 56.0446} C_DIS
LIN {X 83.7505,Y 54.7333,Z 100,A 27.7442,B 24.9245,C -2.0071,E1 25.1348,E2 57.6659} C_DIS
LIN {X 85.8001,Y 51.4626,Z 100,A 25.6109,B 24.9247,C -2.0043,E1 25.1379,E2 59.7951} C_DIS
LIN {X 87.6841,Y 48.182,Z 100,A 23.493,B 24.925,C -2.0003,E1 25.1408,E2 61.9113} C_DIS
LIN {X 89.3377,Y 45.042,Z 100,A 21.2869,B 24.9259,C -1.9879,E1 25.1437,E2 64.1351} C_DIS
LIN {X 91.5329,Y 40.3936,Z 100,A 18.1714,B 24.927,C -1.9727,E1 25.1473,E2 67.2694} C_DIS
LIN {X 92.8499,Y 37.2671,Z 100,A 16.6264,B 24.9263,C -1.9828,E1 25.1489,E2 68.7821} C_DIS
LIN {X 94.1362,Y 33.8862,Z 100,A 14.4653,B 24.927,C -1.9731,E1 25.151,E2 70.9539} C_DIS
LIN {X 95.2125,Y 30.7295,Z 100,A 12.7972,B 24.9267,C -1.9771,E1 25.1524,E2 72.6034} C_DIS
LIN {X 96.1894,Y 27.5204,Z 100,A 10.56,B 24.9281,C -1.9586,E1 25.1542,E2 74.8712} C_DIS
LIN {X 97.7126,Y 21.4941,Z 100,A 7.3198,B 24.9279,C -1.9604,E1 25.1563,E2 78.0885} C_DIS
LIN {X 98.499,Y 17.5411,Z 100,A 4.6924,B 24.9294,C -1.9405,E1 25.1577,E2 80.7476} C_DIS
LIN {X 99.0509,Y 14.0936,Z 100,A 2.403,B 24.9307,C -1.9226,E1 25.1586,E2 83.0657} C_DIS
LIN {X 99.5367,Y 10.1124,Z 100,A 0.9248,B 24.9289,C -1.948,E1 25.159,E2 84.4753} C_DIS
LIN {X 99.7566,Y 7.645,Z 100,A -0.6749,B 24.9297,C -1.9362,E1 25.1594,E2 86.0933} C_DIS
LIN {X 100.0112,Y 2.7513,Z 100,A -3.8811,B 24.9315,C -1.9111,E1 25.1598,E2 89.3395} C_DIS
LIN {X 100.0476,Y -0.4801,Z 100,A -4.9456,B 24.9297,C -1.9367,E1 25.1598,E2 90.3374} C_DIS
LIN {X 100.0012,Y -3.0787,Z 100,A -6.7604,B 24.931,C -1.9188,E1 25.1597,E2 92.1838} C_DIS
LIN {X 99.7292,Y -7.9879,Z 100,A -10.267,B 24.9336,C -1.8821,E1 25.159,E2 95.756} C_DIS
LIN {X 99.2876,Y -12.3278,Z 100,A -11.9025,B 24.9317,C -1.9085,E1 25.1585,E2 97.3196} C_DIS
LIN {X 98.2352,Y -18.9622,Z 100,A -16.7755,B 24.9355,C -1.8551,E1 25.1561,E2 102.2898} C_DIS
LIN {X 97.142,Y -23.9417,Z 100,A -18.6583,B 24.9332,C -1.8872,E1 25.155,E2 104.0862} C_DIS
LIN {X 96.4173,Y -26.7162,Z 100,A -21.1157,B 24.9359,C -1.8494,E1 25.1531,E2 106.6186} C_DIS
LIN {X 95.1842,Y -30.8168,Z 100,A -22.9314,B 24.9347,C -1.8671,E1 25.1516,E2 108.3823} C_DIS
LIN {X 94.0592,Y -34.0973,Z 100,A -24.7889,B 24.9347,C -1.866,E1 25.1499,E2 110.2318} C_DIS
LIN {X 92.8334,Y -37.3078,Z 100,A -27.0338,B 24.9359,C -1.8489,E1 25.1475,E2 112.5047} C_DIS
Enddeposition()
END
